		MesToggleWrite				: BOOL;					(* (NA) Cal: True := read authorised 	*)
		MesToggleRead				: BOOL;					(* (NA) Cal: True := Write authorised	*)
		                                    	                                                	
		
		
		
		
		
		
END_STRUCT
END_TYPE

// ---- 01_Equipement_Library/ProtectRelay/ProtectRelay_PACE100ST.TcDUT
TYPE ProtectRelay_PACE100ST :
STRUCT   
	
		Thermal_Overload			: REAL ; (* %  0 TO 250                         *)
	//Status                                 (*                                     *)
		Comut						: BOOL ; (* Cell's selector is in remote position    *)
		CB_Close					: BOOL ; (*  Cell is closes                                   *)
		CB_In_Alarm					: BOOL ; (*Cell is in alarm                                     *)
		Trip_Counter				: INT;   (*  Number of trip *)

                                  
		Mesdata 					: ProtectRelay;   (*                                     *)
        
END_STRUCT
END_TYPE

// ---- 01_Equipement_Library/ProtectRelay/ProtectRelay_REFIO.TcDUT
TYPE ProtectRelay_REFIO :
STRUCT
	
	MesData				: ProtectRelay ; 	(* Object 								    *)
	MesTransfoAlarm		: BOOL ; 	(* Transfo alarm                              *)
	MesSWOpened			: BOOL ;	(* Sectionneur de ligne ouvert              *)
	MesSWClosed			: BOOL ; 	(* Sectionneur de ligne fermé               *)
	MesEarth			: BOOL ; 	(* Earthing                                 *)
	MesSF6Low			: BOOL ; 	(* SF6 gaz is low                           *)
	MesSF6Unsufficient	: BOOL ; 	(* Sf6  is unsufficient                     *)
	MesTransfoWarning	: BOOL ; 	(* Transfo warning                            *)
	MesOpened			: BOOL ; 	(* Disjoncteur opened                       *)
	MesClosed			: BOOL ; 	(* Disjoncteur is closed                    *)
	MesComutLocal		: BOOL ; 	(* Commutateur Local/Distant.               *)
	
	
END_STRUCT
END_TYPE

// ---- 01_Equipement_Library/ProtectRelay/ProtectRelay_S42.TcDUT
TYPE ProtectRelay_S42 :
STRUCT
	
	MesData							: ProtectRelay ; 	(* Object *)

	MesAlarm_Phase1					: BOOL ;(* Default Phase 1*)		
	MesAlarm_Phase2				    : BOOL ;(*Default Phase 2*)
	MesAlarm_Phase3				    : BOOL ;(*Default Phase 3*)
	MesAlarm_PhaseRpt			    : BOOL ;(*Default Phase RPT (relai presence tension ? ) *)
	MesAlarm_Ground				    : BOOL ;(*Default Ground*)
	MesAlarm_GroundRpt			    : BOOL ;(*Default Ground RPT (relai presence tension ? )*)
	MesAlarm_MaxUInverse			: BOOL ;(*Default Max UI Inverse*)
	MesAlarm_MaxP				    : BOOL ;(*Default Max P *)
	MesAlarm_CB		   			 	: BOOL ;(*Default Circuit breaker *)
	MesAlarm_Watchdog				: BOOL ;(* Défault watchdog*)						
	OUT_CmdOpen	   			 		: BOOL ;(* Circuit breaker Open Command*)
	OUT_CmdClose	    			: BOOL ;(*Circuit breaker Close Command*) 
                      
	MesU0					    	: REAL ;(*(V) Residual Voltage*)
	MesP							: REAL ;(*(kW) Active Power*)
	MesQ							: REAL ;(*(kVAr) Reactive Power*)
	MesCosPhi						: REAL ;(*(p.u) CospPhi*)
	
	MesAlarm_CablesOvercharge 		: BOOL; (*Cables Overcharge*) 		
    MesAlarm_FaultFrom225kV			: BOOL; (*Fault From 225 kV*)		
	
	
END_STRUCT
END_TYPE

// ---- 01_Equipement_Library/ProtectRelay/ProtectRelay_S48.TcDUT
///////////
// Structure For I35. Main Operating Data to be saved ( ex: OPC ) .  
//////////
TYPE ProtectRelay_S48 :
STRUCT
	
		MesData						: ProtectRelay;			(*	(NA) Protection relay									    *)
                                                        	                                               
		                                    				                                                             
		MesU						: REAL;					(* (V) Average Phase to Phase Voltage                           *)
	                                                    	
		MesV1						: REAL ;        		(* (V) Average Phase to Phase Voltage                           *)
		MesV2						: REAL ;				(* (V) Average Phase to Phase Voltage                           *)
		MesV3						: REAL ;				(* (V) Average Phase to Phase Voltage                           *)
       			                                        	                   
		MesP						: REAL; 				(* (Kw)Power on Grid                                            *)
		MesQ						: REAL;					(* (kvar) Power on grid                                         *)
		MesS						: REAL;					(* (KVA) Power apparent                                         *)
		MesCosPhi					: REAL;					(* (NA) power factor                                            *)
		MesTanPhi					: REAL; 				(* (NA) Cal : tan Phi                                           *)
		   

                                 			                                                        
		MesStopPP_UminLong			: BOOL; 				(* (NA) PP is stopping during 2min, because of Long GTE fault	*)
		                                    			                                                          
		EActProd					: REAL; 				(* (MWh) Active Energy Produced                                 *)
		EActCons					: REAL; 				(* (MWh) Active Energy Consummed                                *)
		EReactProd					: REAL; 				(* (MVArh) Reactive Energy Produced                             *)
		EReactCons					: REAL; 				(* (MVArh) Reactive Energy Consummed                            *)
		                                    			                                                           
	// Relais Input                         			
		Input11						: BOOL;					(* (NA) Input 11 du relais de protection                        *)
		Input12                     : BOOL;					(* (NA) Input 12 du relais de protection                        *)
		Input13                     : BOOL;					(* (NA) Input 13 du relais de protection                        *)
		Input14                     : BOOL;					(* (NA) Input 14 du relais de protection                        *)
		Input21						: BOOL;					(* (NA) Input 21 du relais de protection                        *)
		Input22						: BOOL;					(* (NA) Input 22 du relais de protection                        *)
		Input23						: BOOL;					(* (NA) Input 23 du relais de protection                        *)
		Input24						: BOOL;					(* (NA) Input 24 du relais de protection                        *)
		Input25						: BOOL;					(* (NA) Input 25 du relais de protection                        *)
		Input26						: BOOL;					(* (NA) Input 26 du relais de protection                        *)
		
				
END_STRUCT
END_TYPE

// ---- 01_Equipement_Library/ProtectRelay/ProtectRelay_T20.TcDUT
///////////
// Structure For I35. Main Operating Data to be saved ( ex: OPC ) .  
//////////
TYPE ProtectRelay_T20 :
STRUCT
	// I35 Data measures
	
		MesData						: ProtectRelay; (*							*)							
                                           			(*                          *)
	                                       			(*                          *)
		MesFreq						: REAL;			(* (Hz) Frequence of grid   *)
		MesP						: REAL;			(* (Kw)Power on Grid        *)
		MesQ						: REAL;			(* (kvar) Power on grid     *)
		MesS						: REAL;			(* (KVA) Power apparent     *)
		                                   			(*                          *)
		MesTripProtec				: REAL;			(* A                        *)
		MesGlobalWarming		    : REAL;			(* % Au warming of TR       *)


END_STRUCT
END_TYPE

// ---- 01_Equipement_Library/ProtectRelay/ProtectRelay_T87.TcDUT
TYPE ProtectRelay_T87 :
STRUCT
	
	MesData							: ProtectRelay ; 		(* Object 								    *)

	MesAlarm_DiscordSectLigneHTB	: BOOL;   				(*DiscordSectLigneHTB*)
	MesAlarm_DiscordSectMaltHTB		: BOOL;   				(*DiscordSectMaltHTB	*)
	MesAlarm_DiscordSectDisjHTB		: BOOL;   				(*DiscordSectDisjHTB	*)
	MesAlarm_TeleCondamne			: BOOL;   				(*TeleCondamne		*)
	MesAlarm_DeTeleCondamne			: BOOL;   				(*DeTeleCondamne		*)
	MesAlarm_DiscordTeleCondamne	: BOOL;	  				(*DiscordTeleCondamne*)
                                                			
	MesAlarm_IoMaxCoteProd			: BOOL;   				(*IoMaxCoteProd*)
	MesAlarmUMax					: BOOL;   				(*UMax		*)
	MesAlarmUMax_Long				: BOOL;   				(*UMax_Long	*)
	MesAlarm_PhaseRpt				: BOOL;					(*PhaseRpt*)
	MesWarning_ImgTherm				: BOOL;					(*ImgTherm alarm*)
	MesAlarm_ImgTherm				: BOOL;					(*ImgTherm warning*)
	MesAlarm_DifferTransfo			: BOOL;					(*DifferTransfo*)
	MesAlarm_FreqMax				: BOOL;					(*FreqMax*)
	MesAlarm_FreqMin				: BOOL;					(*FreqMin*)	
	                                            			
	MesU0							: REAL;					(*(V) Residual Voltage*)
	MesP							: REAL;					(*(kW) Active Power*)	
	MesQ							: REAL;					(*(kVAr) Reactive Power*)
	

	
END_STRUCT
END_TYPE

// ---- 01_Equipement_Library/ProtectRelay/ProtectRelay_VIP410.TcDUT
TYPE ProtectRelay_VIP410 :
STRUCT
		MesData						: ProtectRelay; 	(* (NA) MesData 																												*)
		MesStatCom					: BOOL ; 			(* (NA) False: device did not respond successfully to most recent read or write request, True: device is responding normally	*)
		MesAvgI1					: REAL ; 			(* (A) Phase 1 Average current                                                                                       			*)
		MesAvgI2					: REAL ; 			(* (A) Phase 2 Average current                                                                                       			*)
		MesAvgI3					: REAL ; 			(* (A) Phase 3 Average current                                                                                       			*)
		MesI0Fault					: REAL ; 			(* (A) Fault current                                                                                                 			*)
		StatusWord					: WORD ; 			(* (NA) Status Word                                                                                                     		*)
		ControlWord					: WORD ; 			(* (NA) Control Word                                                                                                    		*)
END_STRUCT
END_TYPE

// ---- 01_Equipement_Library/ProtectRelay/ProtectRelay_WIP1.TcDUT
///////////
// Structure For I35. Main Operating Data to be saved ( ex: OPC ) .  
//////////
TYPE ProtectRelay_WIP1 :
STRUCT
	// I35 Data measures
	MesData					: ProtectRelay ; (**)


	
END_STRUCT
END_TYPE

// ---- 01_Equipement_Library/Router/Router.TcDUT
TYPE Router :
STRUCT
		MesWatchdog	        : BOOL ; 	(* Watchdog*)
		
		MesAlarmCode		: WORD ;	(* (NA) Internal Akuo AlarmCode		*)
		MesWarningCode		: WORD ; 	(* (NA) Internal Akuo WarningCode   *)
		MesEventCode		: WORD ; 	(* (NA) Internal Akuo EventCode	    *)
		
END_STRUCT
END_TYPE

// ---- 01_Equipement_Library/Router/Router_Standard.TcDUT
TYPE Router_Standard :
STRUCT
		MesData				: Router ;  (* Object *)

		
END_STRUCT
END_TYPE

// ---- 01_Equipement_Library/Sensors/ANA/ANA.TcDUT
TYPE ANA :
STRUCT
	Value 					: REAL ;	(* (-) Analogic Value 					*)
	                                    
	MesAlarmCode			: WORD ;	(* (NA) Internal Akuo AlarmCode     *)
	MesWarningCode			: WORD ;    (* (NA) Internal Akuo WarningCode   *)
	MesEventCode			: WORD ;    (* (NA) Internal Akuo EventCode		*)

END_STRUCT
END_TYPE

// ---- 01_Equipement_Library/Sensors/COM/AllInOne.TcDUT
TYPE AllInOne :
STRUCT
	
	MesWindSp 			: REAL ;		(* (m/s)	 Wind speed measurement of the weather station												        *)
	MesWindDir 			: REAL ;		(* (°) 		 Wind direction measurement of the weather station                                                  *)
	MesHygro			: REAL ;		(* (%) 		 Humidity measurement of the weather station                                                        *)
	MesTemp_Amb 			: REAL ;		(* (°C)		 Ambiant temperature measurement of the weather station                                             *)
	MesDewPoint			: REAL ;		(* (%) 		 Dew point measure of weather station                                                               *)
	MesRain1			: REAL ;		(* (count/h) Rain rate                                                                                          *)
	MesRain2			: REAL ;		(* (count/h) Rain rate                                                                                          *)
	MesRain3			: REAL ;		(* (count/h) Rain rate                                                                                          *)
                                        (*                                                                                                              *)
	MesAlarmWindSp		: REAL ;		(* Alarm for the Wind speed : 0=OFF, 1 = Lower threshold, 2 = Higher threshold                                  *)
	MesAlarmWindDir		: REAL ;		(* Alarm for the Wind direction : 0=OFF, 1 = Lower threshold, 2 = Higher threshold                              *)
	MesAlarmTemp		: REAL ;		(* Alarm for the temp sensor : 0=OFF, 1 = Lower threshold, 2 = Higher threshold                                 *)
	MesAlarmHygro		: REAL ;		(* Alarm for the humidity sensor : 0=OFF, 1 = Lower threshold, 2 = Higher threshold                             *)
	MesAlarmDewPt		: REAL ;		(* Alarm for the dew point sensor : 0=OFF, 1 = Lower threshold, 2 = Higher threshold                            *)
	MesAlarmRain1		: REAL ;		(* Alarm for the rain sensor : 0=OFF, 1 = Lower threshold, 2 = Higher threshold                                 *)
	MesAlarmRain2		: REAL ;		(* Alarm for the rain sensor : 0=OFF, 1 = Lower threshold, 2 = Higher threshold                                 *)
	MesAlarmRain3		: REAL ;		(* Alarm for the rain sensor : 0=OFF, 1 = Lower threshold, 2 = Higher threshold                                 *)
	                                    (*                                                                                                              *)
	MesAlarmCode		: WORD ;  	    (*                                                                                                              *)
	MesWarningCode		: WORD ;  	    (*                                                                                                              *)
	MesEventCode		: WORD ; 	    (*                                                                                                              *)
	
END_STRUCT
END_TYPE

// ---- 01_Equipement_Library/Sensors/COM/SMP1X.TcDUT
TYPE SMP1X :
STRUCT
	
	Value 						: REAL ;		(* (W/m²) Irradiance OF the pyranometer															*)
	Alarm						: REAL ;		(* Alarm for solar radiation (0=Off, 1 = Lower threshold, 2=Higher threshold)                   *)
	Description					: STRING ; 		(* Position and comments on the pyranometer                                                     *)
	                                            (*                                                                                              *)
	MesAlarmCode				: WORD ;  	    (*                                                                                              *)
	MesWarningCode				: WORD ;  	    (*                                                                                              *)
	MesEventCode				: WORD ; 	    (*                                                                                              *)
	
END_STRUCT
END_TYPE

// ---- 01_Equipement_Library/Sensors/TOR/TOR.TcDUT
TYPE TOR :
STRUCT
	
	MesAlarmState 		 		: BOOL  ;		(* TRUE = ALARM													*)
	MesCountAlarm				: UDINT ; 		(* Count the number of time the alarm has been triggered.       *)
                                                (*                                                              *)
	MesAlarmCode				: WORD ;		(* (NA) Internal Akuo AlarmCode                                 *)
	MesWarningCode				: WORD ;   	 	(* (NA) Internal Akuo WarningCode                               *)
	MesEventCode				: WORD ;	 	(* (NA) Internal Akuo EventCode		                            *)

END_STRUCT		
END_TYPE

// ---- 01_Equipement_Library/Sensors/TOR/TOR_Rain.TcDUT
TYPE TOR_Rain :
STRUCT
	
	MesData					: TOR ;		(* MesData 											 *)
	MesRainFall_LastHour  	: REAL;   	(* (mm)Amount of water fall during the last hour	 *)
	MesRainFall_LastDay   	: REAL;   	(* (mm)Amount of water fall during the last Day (mm) *)
	MesRainFall_LastMonth 	: REAL;   	(* (mm)Amour of water fall during the last Year (mm) *)
	                           
	AvgmmHour	  			: REAL; 	(* (mm)Hourly AVG of water fall                      *)
	AvgmmDay   				: REAL;     (* (mm)Daily AVG of water fall                       *)
	AvgmmMonth 				: REAL;     (* (mm) Monthly AVG of water fall                    *)
	
END_STRUCT
END_TYPE

// ---- 01_Equipement_Library/Sensors/TOR/TOR_Standard.TcDUT
TYPE TOR_Standard :
STRUCT
	
	MesData					: TOR ;		(* MesData 											 *)

END_STRUCT		
END_TYPE

// ---- 01_Equipement_Library/Tariff Meter/EM.TcDUT
TYPE EM :
STRUCT
	
	MesEActCons				: REAL ; 		(* Value of Active Energy consumed		*)
	MesEActProd				: REAL ;		(* Value of Active Energy produced      *)
	MesEReactCons			: REAL ;		(* Value of Reactive Energy consumed    *)
	MesEReactProd			: REAL ;		(* Value of Reactive Energy produced    *)
	                                                                             
	MesAlarmCode			: WORD ;	 	(* (NA) Internal Akuo AlarmCode         *)
	MesWarningCode			: WORD ; 		(* (NA) Internal Akuo WarningCode       *)
	MesEventCode			: WORD ; 		(* (NA) Internal Akuo EventCode	        *)

END_STRUCT
END_TYPE

// ---- 01_Equipement_Library/Tariff Meter/EM_Standard.TcDUT
TYPE EM_Standard :
STRUCT
	
	MesData			: EM ; 

END_STRUCT
END_TYPE

// ---- 01_Equipement_Library/Transfo/Transfo.TcDUT
TYPE Transfo :
STRUCT
    MesWarningTemp				: BOOL ;	(* Transfo Temperature warning		    *)
    MesAlarmTemp				: BOOL ;	(* Transfo Temperature Alarm		    *)
    MesAlarmGas					: BOOL ;	(* Transfo Gas Alarm			        *)
    MesAlarmOilLevel			: BOOL ;	(* Transfo Oil Level Alarm		        *)
    MesAlarmsSynthesis			: BOOL ;	(* Transfo Synthesis Alarm              *)
                                                                             
	MesAlarmCode				: WORD ;  	(* (NA) Internal Akuo AlarmCode         *)
	MesWarningCode				: WORD ; 	(* (NA) Internal Akuo WarningCode       *)
	MesEventCode				: WORD ; 	(* (NA) Internal Akuo EventCode	        *)

END_STRUCT
END_TYPE

// ---- 01_Equipement_Library/Transfo/Transfo_HV.TcDUT
TYPE Transfo_HV :
STRUCT

	MesData						: Transfo ; (* Transfo*)

	MesWarningGas					: BOOL  ; (* Buchholz warning*)

	MesWarning_TempLevel1			: BOOL  ; (*ImgTherm1erStade*)
	MesWarning_TempLevel2			: BOOL  ; (*ImgTherm2ndStade*)
	MesTrigger_Deletion				: BOOL  ; (*TransfoDcltSurpression*)

	MesTransfoRefrigLocal			: BOOL  ; (*TransfoRefrigLocal*)
	
	MesTrigger_NonReturnValve		: BOOL  ; (*declenchement clapet anti retour*)
	MesTrigger_ProtectRelay			: BOOL  ; (*DcltRelaisProtectRegl*)
	MesAlarm_TapChanger				: BOOL  ; (*Fault TapChanger*)
	
	


END_STRUCT
END_TYPE

// ---- 01_Equipement_Library/Transfo/Transfo_MV.TcDUT
TYPE Transfo_MV :
STRUCT
	
	MesData						: Transfo ; (* MesData *)


END_STRUCT
END_TYPE

// ---- 01_Equipement_Library/UPS/UPS.TcDUT
///////////
// Structure for UPS. Main Operating Data to be saved (ex: OPC)  
//////////
TYPE UPS :
STRUCT
		MesDischarging				: BOOL ; 			(* (NA) Battery is discharging		*)
		MesAlarm_Ulow				: BOOL ; 			(* (NA) Battery is almost empty     *)
		MesAlarmState				: BOOL ; 			(* (NA) Fault on the charger        *)
		MesUdc  					: REAL ; 			(* (V) DC Load voltage              *)
       		
		
		MesAlarmCode				: WORD ; 			(* Internal Akuo Alarm Code         *)
		MesWarningCode				: WORD ; 			(* Internal Akuo Warning Code       *)
		MesEventCode				: WORD ; 			(* Internal Akuo Warning Code 	    *)
        
		MesCP_Read					: BOOL := FALSE ;   (* Read function enable             *)
		MesAlarmCom					: BOOL ; 			(* Communication alarm              *)
	
END_STRUCT
END_TYPE

// ---- 01_Equipement_Library/UPS/UPS_CXC.TcDUT
///////////
// Structure For I35. Main Operating Data to be saved ( ex: OPC ) .  
//////////
TYPE UPS_CXC :
STRUCT
	
	MesData				: UPS ; 	(* Object 									*)
	            		            (*                                          *)
	MesU				: REAL ; 	(*(V) AC voltage                            *)
	MesIload			: REAL ; 	(*(A) DC Load current                       *)
	MesUBatt			: REAL ; 	(*(V) Battery voltage                       *)
	MesIBatt			: REAL ; 	(*(A) Battery Current                       *)
	MesSoC  			: REAL ; 	(*(%) Battery SoC                           *)
	MesIdc  			: REAL ; 	(*(A) battery + load Current                *)

	
	MesOverTempBatt 	: BOOL ; 	(* OverTemperature of the battery alarm		*)
	MesCBUpsOpened		: BOOL ; 	(* UPS CB opened alarm                      *)
	
		
	
END_STRUCT
END_TYPE

// ---- 01_Equipement_Library/UPS/UPS_ENERIS.TcDUT
///////////
// Structure For I35. Main Operating Data to be saved (ex: OPC).  
//////////
TYPE UPS_Eneris :
STRUCT
	// I35 Data measures
		MesData                     : UPS;  (* MesData *)
		
END_STRUCT
END_TYPE

// ---- 01_Equipement_Library/UPS/UPS_Eneris.TcDUT
///////////
// Structure For I35. Main Operating Data to be saved (ex: OPC).  
//////////
TYPE UPS_Eneris :
STRUCT
	// I35 Data measures
		MesData                     : UPS;  (* MesData *)
		
END_STRUCT
END_TYPE

// ---- 01_Equipement_Library/UPS/UPS_Eneris.TcDUT
///////////
// Structure For I35. Main Operating Data to be saved (ex: OPC).  
//////////
TYPE UPS_Eneris :
STRUCT
	// I35 Data measures
		MesData                     : UPS;  (* MesData *)
		
END_STRUCT
END_TYPE

// ---- 01_Equipement_Library/UPS/UPS_PS10048.TcDUT
///////////
// Structure for PS100_48. Main operating data to be saved (ex:OPC).  
//////////
TYPE UPS_PS10048 :
STRUCT
		MesData             : UPS; 			(* MesData 																		*)
		                            		                                                                                
		MesSoc				: REAL; 		(* (%) Battery charge indicator 												*)
		MesUdc_48V			: REAL; 		(* (V) 48V output voltage 														*)
		MesUdc_12V			: REAL; 		(* (V) 12V output voltage 														*)
		MesUBatt			: REAL; 		(* (V) 12V battery voltage	    												*)
		MesIdc_12V			: REAL; 		(* (A) 12V output current 														*)
		MesIdc_Bat			: REAL;			(* (A) Battery current 															*)
		                            		                                                                                
		MesDischarge		: REAL; 		(* (V) Serious discharge threshold 												*)
		MesEbackUp			: REAL; 		(* (%) Energy backup threshold 	   												*)
		MesCapacity_Nom		: REAL; 		(* (Ah) NomCapa 				   												*)
		                                                                       												
		MesEBackUpEna		: BOOL;  		(* (Na) Energy backup enabled 	   												*)
		MesBatTestPer		: BOOL;  		(* (Na) Battery test period 	  												*)
		MesVacTripSelect	: BOOL;  		(* (NA) 0: Low. Off = 52Vac, Low = 129Vac. 1: High. Off = 69Vac, Low = 172Vac	*)
		                                                                                                                    
		MesToggleWrite		: BOOL;			(* (NA) Cal : True = read authorised  											*)
		MesToggleRead		: BOOL;			(* (NA) Cal : True = Write authorised 											*)
		                           		                                                                                    
		MesAlarm_AcOff		: BOOL;			(* (NA) True = AC off 															*)
		MesAlarm_GeneralOff	: BOOL;			(* (NA) True = Imminent shutdown 												*)
	//	MesAlarm_LowBat		: BOOL;			(* (NA) True = discharge 														*)
		MesAlarm_AcLow		: BOOL;			(* (NA) True = AC power supply low 												*)
		                                                                                                                    
		MesFault_Minor		: BOOL;			(* (NA) True = Minor fault (overtemp, overcurrent, overvolt) 					*)
		MesFault_Major		: BOOL;			(* (NA) True = Major fault : cannot recover 									*)
		MesFault_Bat		: BOOL;			(* (NA) True = Battery disconnected 											*)
		MesFault_Charger	: BOOL;			(* (NA) True = Charger out of order 											*)
		MesFault_12V		: BOOL;			(* (NA) True = 12V absent 														*)
		MesFault_48V		: BOOL;			(* (NA) True = 48V absent 														*)
		                           	
END_STRUCT
END_TYPE

// ---- 04_Application/IO/IO.TcDUT
TYPE IO :
STRUCT
MesEventCode : ARRAY[1..7] OF WORD ; (*Akuo AlarmCode*)

END_STRUCT
END_TYPE

// ---- 04_Application/IO/ST_AI.TcDUT
TYPE ST_AI :
STRUCT
		Value		  AT %I*	: INT	;
		Description 			: STRING	;

END_STRUCT
END_TYPE

// ---- 04_Application/IO/ST_AO.TcDUT
TYPE ST_AO :
STRUCT
		Value		  AT %Q*	: INT	;
		Description 			: STRING	;

END_STRUCT
END_TYPE

// ---- 04_Application/IO/ST_DI.TcDUT
TYPE ST_DI :
STRUCT
		Value		  AT %I*	: BOOL	;
		Description 			: STRING	;

END_STRUCT
END_TYPE

// ---- 04_Application/IO/ST_DO.TcDUT
TYPE ST_DO :
STRUCT
		Value		  AT %Q*	: BOOL	;
		Description 			: STRING	;

END_STRUCT
END_TYPE

// ---- 00_FunctionsBlocks/Communication/IEC104/GVL_Cst.TcGVL
{attribute 'qualified_only'}
VAR_GLOBAL CONSTANT
		CstNbAOEntries			: INT :=  50 ;
END_VAR

// ---- 00_FunctionsBlocks/Fifo/GVL_Fifo.TcGVL
VAR_GLOBAL CONSTANT 
		Max_buffer_size_G					: UDINT:=10000000; // Max buffer size of fifo
END_VAR

// ---- 04_Application/CONFIG/GVL_BASE.TcGVL
///////////////////////
// DO NOT MODIFY :  
// Maximal number of objects  - Maximal array size 
////////////////////
VAR_GLOBAL CONSTANT 
	// PRODUCT 
	CstNbPTR_G					: BYTE := 4 ;  				// (NA) Number of PTR
	CstNbESS_G   				: BYTE := 3 ;  				// (NA) Number of ESS


	// EQUIPMENT
		//SUB_MV
	CstNbFeederMVCB_G			: BYTE	:= 3 ; 
		// PTR 
	CstNbInv_PTR_G				: BYTE := 2 ;				// Maximal Number of PV Inverters for PTR
	CstNbSB_INV_G				: BYTE := 32 ;				// Maximal Number of String box in inverter

		// EM 		
	CstNbEM_G					: BYTE := 1;				// Number of Energy Meters
		
		//ESS		
	CstNbPcs_ESS				: BYTE := 2  ;
	CstNbPowerCol_PCS_G			: BYTE := 3  ;				// Maximal Number of Power colonne by PCS
	CstNbHvac_ESS				: BYTE := 2  ;
	CstNbBank_Ess				: BYTE := 2  ;
	CstNbRack_BBMS				: BYTE := 2  ;
				
		
		//WS		
	CstNbPyrano					: UINT := 5;
	CstNbAnemo					: UINT := 1;
	CstNbPanTmp					: UINT := 4;
	CstNbAmbTmp					: UINT := 3;	
		
	// PP 
	CstNbCouplermax_G			: BYTE 	:= 100 ;			// Maximal number of ethercat devices 
	CstNbAlarmIO_G				: BYTE := 10 ; // Number of Event in PRG_IO.
	
	
	(*               SMS               							*)
	CstNbUser					: SINT:=10; //Nbr d'utilisateur utilisé par AX_Numtel
	CstNbCMD					: SINT:=20; //Nbr commande utilisé par AX_CMD_SMS
	CstNbAlarmCode				: INT:=213;  //Number of alarmcode use in AlarmManager
	
	// TIMEZONE
	    (* Indonesia East Standard Time Zone settings *)
        FRANCE_TZI : ST_TimeZoneInformation := (bias:=-60,
                                       		 				standardName:='Heure Française',
                                        					standardDate:=(wYear:=0,wMonth:=10,wDayOfWeek:=0,wDay:=27,wHour:=3),
                                        					standardBias:=0,
                                        					daylightName:='None',
                                        					daylightDate:=(wYear:=0,wMonth:=3,wDayOfWeek:=0,wDay:=31,wHour:=2),
                                        					daylightBias:=0);
			
		CstPhoneIndicator_G		: STRING := '+33';
			
		CstCycleTime_G			: INT := 10 ; 			// (ms) Cycle Time of the CPU . 

		CstNbRedundantVariableMax_G	: UINT := 553 ;
		CstNbParamOPCUA				: UINT := 100 ; 
	
END_VAR
VAR_GLOBAL
	sTimeGMT_G          	: STRING;				// Full Date Time for historization (GMT) 
	sTimeLocal_G		 	: STRING ;				// Local Time 
	CalGMTTimeStruct		: TIMESTRUCT ; 			// GMT Time Structure

	ParamOpenVpnFile		: STRING := '';			// Path to openvpn file. 
	ParamIpPublic 			: STRING(255);			// Public IP 
	MesSizeCdrive_PLC		: REAL := 100000 ; 		// (Mo) Remaining Disk space
	MesSizeCdrive_IndusPC	: REAL := 100000 ; 		// (Mo) Remaining Disk space
END_VAR

// ---- 04_Application/CONFIG/GVL_Beckhoff.TcGVL
VAR_GLOBAL
	CalLocalTimeStruct			: TIMESTRUCT;		// Local Time Structure
	CstTimeZone_G				: ST_TimeZoneInformation 	:= WEST_EUROPE_TZI ;	// Local TimeZone
	ParamDirBaseStore		: STRING := 'C:\TwinCAT\Functions\Historisation\';	// Directroy for the historization
	
	

	
END_VAR

// ---- 04_Application/CONFIG/GVL_CFG.TcGVL
///////////////
// Configuration Files. Define Power Plant sizing and references. 
//////////////
VAR_GLOBAL 
		CstPLCBackup 			: BOOL := FALSE ;  			// TRUE if this PLC is used as a backup . 
		CstNetAmsId_Slave		: STRING(20):= '5.49.202.22.1.1'; //NetAMSId Slave .'5.79.170.90.1.1'
		CstNetAmsId_IndusPC		: STRING(20):= ''; // set '' if no Indus PLC
		//CstIPIEC104			: STRING := '10.101.111.1' ; 
		
		
END_VAR
	
VAR_GLOBAL 
	// Solar Classique //
		A1_PP					: FB_PP  ;  								// MCA Power Plant 
 
	// PRODUCT DEFINITION //
		//PTR 
		AX_PTR 					: ARRAY[1..CstNbPTR_G] OF FB_PTR ; 	 		// Array with AMG products
		
		//SUB_MV
		A1_SUBMV				: FB_SUBMV ;	 					 		// SUB_MV		
		
		//WEATHER STATION
		A1_WS					: FB_WS;
		
		//ESS 
		//AX_ESS				: ARRAY[1..CstNbESS_G] OF FB_ESS ; 
		
	// GLOBAL VARIABLE //
	
		CmdClearFault_G			: BOOL ; 									// (NA) Clear all permanent faults
		CmdInit_G				: BOOL ; 									// (NA) Global Init Action
		CstIPIEC104				: STRING := '10.111.109.1' ; 		
END_VAR

// ---- 04_Application/CONFIG/GVL_Check.TcGVL
VAR_GLOBAL
	FaultCheck_G : BOOL ; // Test if Fault 
	Fault_Count_G: CTU  ; // Counter 	
	

END_VAR

// ---- 04_Application/CONFIG/GVL_DataBaseStructures.TcGVL
{attribute 'qualified_only'}
VAR_GLOBAL
	AX_StructModbusTCP 	AT %MW112 	: ARRAY[1..10000] OF WORD;
END_VAR

// ---- 04_Application/CONFIG/GVL_EmulConfig.TcGVL

VAR_GLOBAL CONSTANT 
	ParamVarAdsMax_G				: UINT := 82 ; // Maximum Object to exchange in Ads
END_VAR

VAR_GLOBAL
	
	ParamCycleTime_Emul				: REAL := 10 ; // Temps de reference d'emulation en ms . 

	MesFreqGen 						: REAL := 50;
	MesUGen							: REAL := 20600;
	ParamLossImpedance				: REAL := 0.000004 ; // Ohmic value to account for transfo losses . 2 10^-8 ohm.m * 200 m .
	
	MesP_INVmppt					: REAL := 2500; // MPPT Power for one inverter 
	
	SoCInit							: REAL := 50 ; 
 
	//////   IO ////// 
	MesTempExt: INT;
	MesWindDir: INT;
	MesWindSpd : INT ; 
	MesHygroExt: INT;
	MesPyra		: INT  ;
	// SuBMV 
	
	iCouplerStatePDL				: UINT ; 
	
	MeasureMVCB_Closed						: BOOL := TRUE; 
	MeasureMVCB_Opened						: BOOL ; 
	MeasureMVCB_Fuse						: BOOL ; 
	MeasureMVCB_Malt						: BOOL ; 
	

	MainMVCB_ComutLocal						: BOOL := TRUE; 
	MainMVCB_Malt						: BOOL ; 
	MainMVCB_Close						: BOOL;
	MainMVCB_Open						: BOOL ;
	
	FeederMVCBClose_External			: ARRAY[1..CstNbFeederMVCB_G] OF BOOL ; 
	FeederMVCBOpen_External			: ARRAY[1..CstNbFeederMVCB_G] OF BOOL ; 	

	FeederMVCB_ComutLocal		: ARRAY[1..CstNbFeederMVCB_G] OF BOOL ; 
	FeederMVCB_Malt		: ARRAY[1..CstNbFeederMVCB_G] OF BOOL ; 
	
	PDLEsState1_IO                : BOOL:=TRUE;
	PDLChainBESSState1_IO         : BOOL;
	PDLMainCBAuxState1_IO         : BOOL;
	PDLCB_SourceSwitch1State1_IO	:BOOL := TRUE; 
	PDLCB_SourceSwitch2State1_IO	:BOOL; 
	PDLCB_HTA1State1_IO           : BOOL;
	PDLCB_HTA2State1_IO           : BOOL;
	PDLCB_Rearmement1State1_IO    : BOOL;
	PDLCB_Rearmement2State1_IO    : BOOL;
	PDLIN_MesCbUPS_IO             : BOOL;    
	PDLFireSystemCBFSS_IO         : BOOL;
	PDLDsBTState1_IO              : BOOL;
	PDLDsHTState1_IO              : BOOL;
	PDLUPSFaultSynthesis_IO       : BOOL;  
	PDLUPSDischarging_IO          : BOOL;  
	PDLRPNWatchDog_IO             : BOOL := TRUE ;  
	PDLRPNWatchdogREU615_IO       : BOOL := TRUE  ;  
	PDLRPNAlarmIPos_IO            : BOOL;  
	PDLRPNAlarmVolt_IO				:BOOL; 
	
	PDLFireSystemWarning_IO			: BOOL;
	PDLFireSystemAlarm_IO			: BOOL;
	PDLFireSystemWatchdog_IO		: BOOL;
	
	
	
(*	
	// ESS
	MesTemp							: ARRAY[1..CstNbEss] OF ARRAY[1..4] OF INT;	
	MesHygr							: ARRAY[1..CstNbEss] OF ARRAY[1..4] OF INT;
	MesSpdState						: ARRAY[1..CstNbEss] OF BOOL;
	MesPcsDs						: ARRAY[1..CstNbEss] OF BOOL;
	MesBatDs						: ARRAY[1..CstNbEss] OF BOOL;
	MesToS							: ARRAY[1..CstNbEss] OF BOOL;
	Cb_Q31_Close					: ARRAY[1..CstNbEss] OF BOOL;
	Cb_Q31_Open						: ARRAY[1..CstNbEss] OF BOOL;
	MesPcs1Sd						: ARRAY[1..CstNbEss] OF BOOL;
	MesPcs2Sd						: ARRAY[1..CstNbEss] OF BOOL;
	MesEs							: ARRAY[1..CstNbEss] OF BOOL;
	Ds_Pcs							: ARRAY[1..CstNbEss] OF BOOL;
	Ds_Bat							: ARRAY[1..CstNbEss] OF BOOL;
	CmdReset_IO						: ARRAY[1..CstNbEss] OF BOOL;			
	MesUpsAlarm						: ARRAY[1..CstNbEss] OF BOOL;		
	MesUpsDischarging				: ARRAY[1..CstNbEss] OF BOOL;		
	MesSupplyFlt_40A_RC				: ARRAY[1..CstNbEss] OF BOOL;	
	MesSup_10A_PLC					: ARRAY[1..CstNbEss] OF BOOL;		
	bBatFireWarning					: ARRAY[1..CstNbEss] OF BOOL;
	bBatFireFault					: ARRAY[1..CstNbEss] OF BOOL;
	bBatFireAlarm					: ARRAY[1..CstNbEss] OF BOOL;
 	bDcSwitchBank1 					: ARRAY[1..CstNbEss] OF BOOL;
 	bDcSwitchBank2	 				: ARRAY[1..CstNbEss] OF BOOL;
 	bFanBank1	 					: ARRAY[1..CstNbEss] OF BOOL;
 	bFanBank2	 					: ARRAY[1..CstNbEss] OF BOOL;
	iCouplerState: ARRAY[1..CstNbESS]OF UINT;
	bCmdResetEss	 					: ARRAY[1..CstNbEss] OF BOOL;
	CoeffSuiviSetpointPcs			: REAL := 0.9;						// Pourcentage de suivi de la consigne à chaque pas de temps : si 1, MesPac = SetptP d'un pas de temps à l'autre, si 0 ne suit pas du tout le setpoint

*)
END_VAR

// ---- 04_Application/MAIN/MAIN_Emul.TcPOU
PROGRAM MAIN_Emul
VAR
	TP_1		: TP;
	TP_2		: TP;
	
	ClockReadIO				: BOOL;
	ClockReadCOM			: BOOL;
	//M_INIT VARIABLE //
		bInit					: BOOL := TRUE ;						// Initialization variable

		
		WriteAds		: ADSWRITE;
		bTest			: BOOL;
		
		
		// DATETIME //	
		FB_LocalSystTime      	: FB_LOCALSYSTEMTIME;	// Get time function
		FB_ToGMT : FB_TzSpecificLocalTimeToSystemTime;	// Local to UTC Time function
		TON_Time				: TON;
		CalLocalTimeStruct_Temp: TIMESTRUCT;
		//init
		FB_GetSystemTime        : GETSYSTEMTIME;						// GEt time function
		
		FB_ToLocal 				: FB_FileTimeToTzSpecificLocalTime;		// UTC to local Time function
		fileTime        		: T_FILETIME;							// Filetime format for UTC Time 
		FileTimeLocal			: T_FILETIME;							// Filetime format for local time		
		
		
		
		

END_VAR

VAR_OUTPUT
			OUT_CalRunningPLC_IO 		: BOOL ; 
END_VAR

	TP_1(IN:=NOT TP_1.Q , PT:= T#100MS);		// Pour les IO
	ClockReadIO 		:= TP_1.Q;
	TP_2(IN:=NOT TP_1.Q , PT:= T#1S);		// Pour la com
	ClockReadCOM 		:= TP_2.Q;

// INITIALIZATION//
	IF bInit OR CmdInit_G THEN

		M_Init() ; 
		bInit := FALSE; 
	END_IF
	

	TON_Time(IN:= TRUE, PT:=T#1200MS ) ; 
	FB_LocalSystTime(
		bEnable := TRUE,
		dwCycle := 1,
		systemTime => CalLocalTimeStruct_Temp);

	IF TON_Time.Q THEN 
		CalLocalTimeStruct:= CalLocalTimeStruct_Temp ; 
	END_IF
		
		FB_ToGMT(
		in	:= CalLocalTimeStruct,
		tzInfo := CstTimeZone_G,
		out	=> CalGMTTimeStruct);
	
	sTimeGMT_G	:= SYSTEMTIME_TO_STRING(CalGMTTimeStruct);
	sTimeLocal_G	:= SYSTEMTIME_TO_STRING(CalLocalTimeStruct);	

	
OUT_CalRunningPLC_IO := TRUE ; 

// INPUTS //

	PRG_IO() ; 	// Emul the IO
	PRG_IO.M_Inputs() ;  // On mets à jour les variables emulées pour l'ecriture

// PROGRAMMS CALLS //
		ADS_Custom();	// On execute le read et le write . 
	// Hybrid Power PLant 
		A1_PP();
	
	// Historization //
	PRG_IO.M_Outputs() ;  // On recupère les commandes IO. 
	
// OUTPUTS //

METHOD M_Init : BOOL
VAR_INPUT
END_VAR

VAR 
	Year : STRING ; 
	Month: STRING ; 
	Day : STRING ; 
	Hour: STRING ; 
	Str_Temp: STRING;
END_VAR
//CstCycleTime_G 		:= 50 ;							// Cycle Time
CstTimeZone_G 		:= WEST_EUROPE_TZI ; 		// Local Time Zone 
	



// Get the Windows time ( not accurate ) at startup before updating the system time. 
	// DateTime 
	
	
	FB_GetSystemTime(
		timeLoDW	=> fileTime.dwLowDateTime, 
		timeHiDW	=> fileTime.dwHighDateTime);
		
	FB_ToLocal(
		in			:=fileTime,
		tzInfo 		:= CstTimeZone_G,
		out		 	=> FileTimeLocal);
		
CalLocalTimeStruct := FILETIME_TO_SYSTEMTIME(FileTimelocal) ; 


Year := CONCAT(STR1:= WORD_TO_STRING(CalLocalTimeStruct.wYear), STR2:= '_') ; 
Month := CONCAT(STR1:= WORD_TO_STRING(CalLocalTimeStruct.wMonth), STR2:= '_') ;
Day := CONCAT(STR1:=WORD_TO_STRING(CalLocalTimeStruct.wDay), STR2:= ' ') ;
Hour := CONCAT(STR1:=WORD_TO_STRING(CalLocalTimeStruct.wHour), STR2:= 'h') ;

Str_Temp := Year ; 
Str_Temp := CONCAT(STR1:=Str_Temp , STR2:= Month )  ; 
Str_Temp := CONCAT(STR1:=Str_Temp , STR2:= Day )  ; 	
Str_Temp := CONCAT(STR1:=Str_Temp , STR2:= Hour )  ; 

A1_PP.MesData.MesStartTime 		:= Str_Temp  ; 	// Jour du dernier update de code .
END_METHOD

END_PROGRAM

// ---- 04_Application/IO/PRG_IO.TcPOU
PROGRAM PRG_IO
///////////
// This Program is used as an interface between code variable and the I/O cards
//////////
VAR_INPUT
	
//PP States //
	MesCouplerStateSUBMV		: ST_AI ; 

// EXECUTE VARIABLES //
	IN_CmdInhibOutput_OPC		: BOOL :=TRUE ; 
	
END_VAR
VAR 	
//M_INIT VARIABLES //
	bInit						: BOOL	:=TRUE ;			// Initialization variables
	iTest                       : INT;
END_VAR

VAR_INPUT
	KK : INT ;
	
	MesIO_SUBMV_EL1809_1 : ARRAY [1..16] OF ST_DI ; 
	MesIO_SUBMV_EL1809_2 : ARRAY [1..16] OF ST_DI ; 
	MesIO_SUBMV_EL1809_3 : ARRAY [1..16] OF ST_DI ;
	MesIO_SUBMV_EL1809_14 : ARRAY [1..16] OF ST_DI ; 
	MesIO_SUBMV_EL2809_4 : ARRAY [1..16] OF ST_DO ; 
	MesIO_SUBMV_EL3024_5 : ARRAY [1..4] OF ST_AI ; 
	MesIO_SUBMV_EL3024_12 : ARRAY [1..4]  OF ST_AI ;
	MesIO_SUBMV_EL3024_13 : ARRAY [1..4]  OF ST_AI ;
	MesIO_PTR_1_EL3024_8 : ARRAY [1..4] OF ST_AI ; 
	MesIO_PTR_1_EL1809_9 : ARRAY [1..16] OF ST_DI ; 
	MesIO_PTR_1_EL2809_10 : ARRAY [1..16] OF ST_DO ; 
	MesIO_PTR_2_EL3024_8 : ARRAY [1..4] OF ST_AI ; 
	MesIO_PTR_2_EL1809_9 : ARRAY [1..16] OF ST_DI ; 
	MesIO_PTR_2_EL2809_10 : ARRAY [1..16] OF ST_DO ; 
	MesIO_PTR_3_EL3024_8 : ARRAY [1..4] OF ST_AI ; 
	MesIO_PTR_3_EL1809_9 : ARRAY [1..16] OF ST_DI ; 
	MesIO_PTR_3_EL2809_10 : ARRAY [1..16] OF ST_DO ; 
	
END_VAR

// Initializing the static variables //  
	IF bInit OR CmdInit_G THEN
		M_Init() ; 
		bInit		:= FALSE ; 
	END_IF
	
	// EMULATOR OF IO 
	
	// On met ici les calculs pour émuler des variables IO qui ne serait pas liée à des commandes 

A1_SUBMV.IN_MesCouplerState_IO							:= iCouplerStatePDL ;
A1_SUBMV.A1_MeasureMVCB.IN_CmdExternalClose_Emul 		:=  MeasureMVCB_Closed ; 
A1_SUBMV.A1_MeasureMVCB.IN_CmdExternalOpen_Emul 		:=  MeasureMVCB_Opened ; 

FOR KK:= 1 TO CstNbFeederMVCB_G DO 
	A1_SUBMV.AX_FeederMVCB[KK].IN_CmdExternalClose_Emul := FeederMVCBClose_External[KK] ;
	A1_SUBMV.AX_FeederMVCB[KK].IN_CmdExternalOpen_Emul  := FeederMVCBOpen_External[KK] ;
	A1_SUBMV.AX_FeederMVCB[KK].IN_MesComutLocal_IO 		:=  FeederMVCB_ComutLocal[KK] ; 
	A1_SUBMV.AX_FeederMVCB[KK].IN_MesEarth_IO 			:=  FeederMVCB_Malt[KK]; 
END_FOR

// Close cells 
A1_SUBMV.A1_GridMVCB.IN_CmdExternalClose_Emul 		  := TRUE;
A1_SUBMV.A1_AuxMVCB.IN_CmdExternalClose_Emul   		  := TRUE;
A1_SUBMV.A1_MainMVCB.A1_Sect.IN_CmdExternalClose_Emul := TRUE; 


A1_SUBMV.A1_MeasureMVCB.IN_MesFuse_IO :=  MeasureMVCB_Fuse ; 
A1_SUBMV.A1_MeasureMVCB.IN_MesEarth_IO :=  MeasureMVCB_Malt ; 

IF A1_SUBMV.A1_MainMVCB.ParamComutNc THEN 
	A1_SUBMV.A1_MainMVCB.IN_MesComutLocal_IO :=  NOT MainMVCB_ComutLocal ; 
ELSE
	A1_SUBMV.A1_MainMVCB.IN_MesComutLocal_IO :=   MainMVCB_ComutLocal ;
END_IF

A1_SUBMV.A1_MainMVCB.IN_MesEarth_IO :=  MainMVCB_Malt ; 
A1_SUBMV.A1_MainMVCB.IN_CmdExternalClose_Emul	:= MainMVCB_Close ; 
A1_SUBMV.A1_MainMVCB.IN_CmdExternalOpen_Emul	:= MainMVCB_Open OR PDLRPNAlarmIPos_IO OR PDLRPNAlarmVolt_IO; 

A1_SUBMV.A1_ES_LV.IN_MesState1_IO                    := PDLEsState1_IO                   ;
A1_SUBMV.A1_ES_MV.IN_MesState1_IO                    := PDLEsState1_IO                   ;
A1_SUBMV.A1_MainCB_LV.IN_MesState1_IO                := PDLMainCBAuxState1_IO            ;

A1_SUBMV.A1_UPS_24v.IN_MesCbUPS_IO                   := PDLIN_MesCbUPS_IO                ;    
A1_SUBMV.A1_UPS_48v.IN_MesCbUPS_IO                   := PDLIN_MesCbUPS_IO                ;    

//A1_SUBMV.A1_SAFE_FireSystem.IN_MesCBFSS_IO            := PDLFireSystemCBFSS_IO         ;
A1_SUBMV.A1_DS_LV.IN_MesState1_IO                    := PDLDsBTState1_IO                 ;
A1_SUBMV.A1_DS_MV.IN_MesState1_IO                    := PDLDsHTState1_IO                 ;
A1_SUBMV.A1_UPS_24v.IN_MesFault_IO              	 := PDLUPSFaultSynthesis_IO          ; 
A1_SUBMV.A1_UPS_48v.IN_MesFault_IO              	 := PDLUPSFaultSynthesis_IO          ; 

A1_SUBMV.A1_ProtectRelay.IN_MesWatchDog_IO           := PDLRPNWatchDog_IO                ; 
A1_SUBMV.A1_ProtectRelay.IN_MesWatchDog_IO           := PDLRPNWatchdogREU615_IO          ; 
A1_SUBMV.A1_ProtectRelay.IN_MesAlarmIMax_IO          := PDLRPNAlarmIPos_IO               ; 
A1_SUBMV.A1_ProtectRelay.IN_MesAlarmUmin_IO			 := PDLRPNAlarmVolt_IO				;		

// WS 
A1_WS.A1_Temp_Ext.IN_MesValue1_IO	:= MesTempExt ; 
A1_WS.AX_Temp_Panel[1].IN_MesValue1_IO := MesTempExt;
A1_WS.A1_WindDir.IN_MesValue1_IO	:= MesWindDir ; 
A1_WS.A1_WindSp.IN_MesValue1_IO	:= MesWindSpd ; 

FOR KK:=1 TO CstNbPyrano DO 
	A1_WS.Ax_Pyrano[KK].IN_MesValue1_IO :=  MesPyra ; 
END_FOR 		




// ESS
(*	
FOR KK := 1 TO CstNbEss DO
	AX_ESS[KK].AX_TmpSensors[1].IN_MesValue_IO1 := MesTemp[KK][1];
	AX_ESS[KK].AX_HygroSensors[1].IN_MesValue_IO1 := MesHygr[KK][1];
	
	FOR LL := 2 TO 4 DO
		AX_ESS[KK].AX_TmpSensors[LL].IN_MesValue_IO1 := REAL_TO_INT(AX_ESS[KK].AX_HVAC[1].MesDataExd.MesData.MesTempRoom/50*32767) ; //MesTemp[KK][LL];
		AX_ESS[KK].AX_HygroSensors[LL].IN_MesValue_IO1 := REAL_TO_INT(AX_ESS[KK].AX_HVAC[1].MesDataExd.MesData.MesHygroAmb/100*32767) ;// MesHygr[KK][LL];
		
	END_FOR
	//MesIoESS_DI_1[KK][4].Value := GVL_EmulConfig.MesSpdState[KK];
	
	
	AX_Ess[KK].A1_Spd.IN_MesState1_IO 								:= 	MesSpdState[KK];						
	AX_ESS[KK].A1_Ds_Pcs.IN_MesState1_IO 							:=  MesPcsDs[KK];								
	AX_ESS[KK].A1_Ds_Bat.IN_MesState1_IO 							:=  MesBatDs[KK];								
	AX_ESS[KK].A1_ToS.IN_MesState1_IO 								:=  MesToS[KK];								
	AX_ESS[KK].A1_Cb_Q31.IN_CmdExternalClose_Emul							:=  Cb_Q31_Close[KK];							
	AX_ESS[KK].A1_Cb_Q31.IN_CmdExternalOpen_Emul 							:=  Cb_Q31_Open[KK];							
	AX_ESS[KK].A1_Sd_Pcs.IN_MesState1_IO 							:=  MesPcs1Sd[KK];							
	AX_ESS[KK].A1_Sd_Pcs.IN_MesState2_IO 							:=  MesPcs2Sd[KK];							
//	AX_ESS[KK].A1_Sd_Bat.IN_MesState1_IO 							:=  MesBat1Sd[KK];							
	AX_ESS[KK].A1_Es.IN_MesState1_IO 								:=  MesEs[KK];										
	AX_ESS[KK].A1_Ds_Pcs.IN_MesState1_IO 							:=  Ds_Pcs[KK];						
//	AX_ESS[KK].A1_Fuse1_Cab1.IN_MesState1_IO 						:=  Fuse1_Cab1[KK];						
//	AX_ESS[KK].A1_Fuse2_Cab1.IN_MesState1_IO 						:=  Fuse2_Cab1[KK];						
	AX_ESS[KK].A1_Ds_Bat.IN_MesState1_IO 							:=  Ds_Bat[KK];						
//	AX_ESS[KK].A1_Fuse1_Cab2.IN_MesState1_IO  						:=  Fuse1_Cab2[KK];						
//	AX_ESS[KK].A1_Fuse2_Cab2.IN_MesState1_IO  						:=  Fuse2_Cab2[KK];					
	AX_ESS[KK].IN_CmdReset_IO 										:=  CmdReset_IO[KK];				
	AX_ESS[KK].A1_UPS.IN_MesFaultSynthesis_IO						:=  MesUpsAlarm[KK];	
	AX_ESS[KK].A1_UPS.IN_MesDischarging_IO							:=  MesUpsDischarging[KK] ; 				
	AX_ESS[KK].A1_CB_PLC24V.IN_MesState1_IO					 		:=  MesSup_10A_PLC[KK];			
	AX_ESS[KK].A1_CB_RackCtrl24V.IN_MesState1_IO					:=  MesSupplyFlt_40A_RC[KK];			
	AX_ESS[KK].A1_FSS.IN_MesWarning_IO					 			:=  bBatFireWarning[KK];		
	AX_ESS[KK].A1_FSS.IN_MesFault_IO					 			:=  bBatFireFault[KK];	
	AX_ESS[KK].A1_FSS.IN_MesAlarm_IO					 			:=  bBatFireAlarm[KK];		
	AX_ESS[KK].AX_CB_ChainDcSwitchBank[1].IN_MesState1_IO           :=  bDcSwitchBank1[KK];		     
	AX_ESS[KK].AX_CB_ChainDcSwitchBank[2].IN_MesState1_IO           :=  bDcSwitchBank2[KK];	
	AX_ESS[KK].AX_CB_ChainFanBank[1].IN_MesState1_IO                :=  bFanBank1[KK];		     
	AX_ESS[KK].AX_CB_ChainFanBank[2].IN_MesState1_IO                :=  bFanBank2[KK];	   
	AX_ESS[KK].IN_MesCouplerState_IO								:= iCouplerState[KK] ;
	AX_ESS[KK].IN_CmdReset_IO										:= bCmdResetEss[KK] ; 	


END_FOR

	
*)

METHOD M_Init : BOOL
VAR
	KK : BYTE;
	
	LL: UINT ; 
	MM: INT;
	JJ: INT;
	
END_VAR

// WS
	MesTempExt	:= 16000 ; 
	MesWindDir     := 16000 ; 
	MesWindSpd     := 16000 ; 
	MesHygroExt	:= 16000 ; 
	MesPyra		:= 16000 ; 
// 
(*

FOR KK:= 1 TO CstNbESS_G DO 
	FOR LL:= 1 TO CstNbBank_Ess DO 
		FOR MM := 1 TO AX_ESS[KK].AX_Bbms[LL].ParamNbRacks DO
			FOR JJ := 1 TO AX_ESS[KK].AX_Bbms[LL].ParamNbRackString DO 
				MEMCPY(destAddr := ADR(AX_ESS[KK].AX_Bbms[LL].Rea.MesDataExd.MesData.AX_Rack[KK].AX_RACKSTRING[JJ].MesSoC) , srcAddr := ADR(SoCInit) , n:= SIZEOF(SoCInit)) ; 
			END_FOR
		END_FOR
	END_FOR
END_FOR


iCouplerStatePDL :=  8 ; 

PDLChainBESSState1_IO := TRUE ;
FOR KK := 1 TO CstNbEss DO
	FOR LL := 1 TO 4 DO
			 MesTemp[KK][LL] := 16000 ;		//32767 ma value 
			MesHygr[KK][LL] := 16000;
		
	END_FOR
	//MesIoESS_DI_1[KK][4].Value := GVL_EmulConfig.MesSpdState[KK];
	
	
MesSpdState[KK]					:= FALSE ;			
MesPcsDs[KK]					:= FALSE ;				
MesBatDs[KK]					:= FALSE ;				
MesToS[KK]						:= TRUE ;			
Cb_Q31_Close[KK]				:= TRUE ;				
Cb_Q31_Open[KK]					:= FALSE ;				
MesPcs1Sd[KK]					:= FALSE ;			
MesPcs2Sd[KK]					:= FALSE ;			
MesEs[KK]						:= FALSE ;					
Ds_Pcs[KK]						:= FALSE ;	
Ds_Bat[KK]						:= FALSE ;	
CmdReset_IO[KK]					:= FALSE ;	
MesUpsAlarm[KK]	        		:= FALSE ;
MesUpsDischarging[KK] 			:= FALSE ;			
MesSup_10A_PLC[KK]				:= TRUE ;
MesSupplyFlt_40A_RC[KK]			:= TRUE ;		
bBatFireWarning[KK]				:= FALSE ;
bBatFireFault[KK]        		:= FALSE ;
bBatFireAlarm[KK]	    		:= FALSE ;
bDcSwitchBank1[KK]	    		:= FALSE ; 
bDcSwitchBank2[KK]      	 	:= FALSE ;
bFanBank1[KK]		        	:= TRUE ;
bFanBank2[KK]   				:= TRUE ;
iCouplerState[KK]				:= 8 ;
END_FOR
		*)
END_METHOD

METHOD M_Inputs
///////////
// Intput interface between POUs and I/O Cards
//////////////

VAR 
KK							: BYTE ; 					// For LOOP 
MesCouplerStateSUB_MV			: ST_AI ; 
END_VAR

MesIO_SUBMV_EL1809_1[ 1].value  			:= A1_SUBMV.AX_FeederMVCB[1].IN_MesOpened_IO 	;	
MesIO_SUBMV_EL1809_1[ 2].value        		:=   A1_SUBMV.AX_FeederMVCB[2].IN_MesOpened_IO	;
MesIO_SUBMV_EL1809_1[ 3].value        	:=   A1_SUBMV.AX_FeederMVCB[3].IN_MesOpened_IO	;	
MesIO_SUBMV_EL1809_1[ 4].value        		:=   A1_SUBMV.A1_MainMVCB.IN_MesOpened_IO		;
MesIO_SUBMV_EL1809_1[ 5].value        		:=   A1_SUBMV.A1_MainMVCB.IN_MesTripped_IO		;
MesIO_SUBMV_EL1809_1[ 6].value        		:=   A1_SUBMV.A1_MainMVCB.IN_MesEarth_IO  		;
MesIO_SUBMV_EL1809_1[ 7].value        		:=   A1_SUBMV.A1_MainMVCB.IN_MesComutLocal_IO	;
MesIO_SUBMV_EL1809_1[ 8].value        		:=   A1_SUBMV.A1_MainMVCB.IN_MesAlarmPwr_IO		;
MesIO_SUBMV_EL1809_1[ 9].value        		:=   A1_SUBMV.AX_FeederMVCB[1].IN_MesTripped_IO	;
MesIO_SUBMV_EL1809_1[ 10].value    			:=   A1_SUBMV.AX_FeederMVCB[2].IN_MesTripped_IO	;	
MesIO_SUBMV_EL1809_1[ 11].value    		:=   A1_SUBMV.AX_FeederMVCB[3].IN_MesTripped_IO	;  
MesIO_SUBMV_EL1809_1[ 12].value    			:=   A1_SUBMV.AX_FeederMVCB[1].IN_MesAlarmPwr_IO;  	
MesIO_SUBMV_EL1809_1[ 13].value    			:=   A1_SUBMV.AX_FeederMVCB[2].IN_MesAlarmPwr_IO;  	
MesIO_SUBMV_EL1809_1[ 14].value    		:=   A1_SUBMV.AX_FeederMVCB[3].IN_MesAlarmPwr_IO;  
MesIO_SUBMV_EL1809_1[ 15].value    			:=   A1_SUBMV.AX_FeederMVCB[1].IN_MesEarth_IO	;  
MesIO_SUBMV_EL1809_1[ 16].value    			:=   A1_SUBMV.AX_FeederMVCB[2].IN_MesEarth_IO	;  
MesIO_SUBMV_EL1809_2[ 1].value     		:=   A1_SUBMV.AX_FeederMVCB[3].IN_MesEarth_IO	;  
MesIO_SUBMV_EL1809_2[ 2].value     			:=   A1_SUBMV.AX_FeederMVCB[1].IN_MesComutLocal_IO;   
MesIO_SUBMV_EL1809_2[ 3].value     			:=   A1_SUBMV.AX_FeederMVCB[2].IN_MesComutLocal_IO;   
MesIO_SUBMV_EL1809_2[ 4].value    		:= A1_SUBMV.AX_FeederMVCB[3].IN_MesComutLocal_IO ;
MesIO_SUBMV_EL1809_2[ 5].value       		:=   A1_SUBMV.A1_GridMVCB.IN_MesOpened_IO			 ;		
MesIO_SUBMV_EL1809_2[ 6].value       		:=   A1_SUBMV.A1_MeasureMVCB.IN_MesOpened_IO		 ;		
MesIO_SUBMV_EL1809_2[ 7].value       		:=   A1_SUBMV.A1_MeasureMVCB.IN_MesFuse_IO  		 ;		
MesIO_SUBMV_EL1809_2[ 8].value       		:=   A1_SUBMV.A1_MeasureMVCB.IN_MesEarth_IO 		 ;		
MesIO_SUBMV_EL1809_2[ 9].value       		:=   A1_SUBMV.A1_AuxMVCB.IN_MesOpened_IO			 ; 			
MesIO_SUBMV_EL1809_2[ 10].value       		:=   A1_SUBMV.A1_AuxMVCB.IN_MesFuse_IO				 ;
MesIO_SUBMV_EL1809_2[ 11].value       		:=   A1_SUBMV.A1_AuxMVCB.IN_MesEarth_IO				 ;
MesIO_SUBMV_EL1809_2[ 12].value       		:=   A1_SUBMV.A1_ES_LV.IN_MesState1_IO				 ;
MesIO_SUBMV_EL1809_2[ 13].value       		:=   A1_SUBMV.A1_ES_MV.IN_MesState1_IO				 ;
MesIO_SUBMV_EL1809_2[ 14].value       		:=   A1_SUBMV.A1_SD_LV.IN_MesState1_IO				 ;
MesIO_SUBMV_EL1809_2[ 15].value       		:=   A1_SUBMV.A1_SD_MV.IN_MesState1_IO				 ;
MesIO_SUBMV_EL1809_2[ 16].value       		:=   A1_SUBMV.A1_Transfo_Aux.IN_MesAlarmsSynthesis_IO;
MesIO_SUBMV_EL1809_3[ 1].value 				:= 	 A1_SUBMV.A1_MainMVCB.A1_Sect.IN_MesClosed_IO 	 ;    
MesIO_SUBMV_EL1809_3[ 2].value       		:=   A1_SUBMV.A1_Transfo_Aux.IN_MesAlarmGas_IO		 ; 
MesIO_SUBMV_EL1809_3[ 3].value       		:=   A1_SUBMV.A1_Transfo_Aux.IN_MesWarningTemp_IO	 ; 
MesIO_SUBMV_EL1809_3[ 4].value       		:=   A1_SUBMV.A1_Transfo_Aux.IN_MesAlarmTemp_IO		 ; 
MesIO_SUBMV_EL1809_3[ 5].value       		:=   A1_SUBMV.A1_UPS_24v.IN_MesDischarging_IO		 ; 
MesIO_SUBMV_EL1809_3[ 6].value       		:=   A1_SUBMV.A1_UPS_24v.IN_MesFault_IO				 ; 
MesIO_SUBMV_EL1809_3[ 7].value       		:=   A1_SUBMV.A1_UPS_24v.IN_MesBatLow_IO			 ; 
MesIO_SUBMV_EL1809_3[ 8].value       		:=   A1_SUBMV.A1_ProtectRelay.IN_MesAlarmIMax_IO	 ; 
MesIO_SUBMV_EL1809_14[ 6].value       		:=   A1_SUBMV.A1_ProtectRelay.IN_MesAlarmUmin_IO	 ; 
MesIO_SUBMV_EL3024_5[ 1].value       		:=   A1_WS.Ax_Pyrano[1].IN_MesValue1_IO				 ; 
MesIO_SUBMV_EL3024_5[ 2].value       		:=   A1_WS.Ax_Pyrano[2].IN_MesValue1_IO				 ; 
MesIO_SUBMV_EL3024_5[ 3].value       		:=   A1_WS.A1_Temp_Ext.IN_MesValue1_IO				 ; 
MesIO_SUBMV_EL3024_5[ 4].value       		:=   A1_WS.A1_Hygro_Ext.IN_MesValue1_IO				 ; 
MesIO_SUBMV_EL3024_13[ 1].value       		:=   A1_WS.A1_WindDir.IN_MesValue1_IO				 ; 
MesIO_SUBMV_EL3024_13[ 2].value       		:=   A1_WS.A1_WindSp.IN_MesValue1_IO				 ; 
MesIO_PTR_1_EL3024_8[ 1].value       		:=   A1_WS.AX_Temp_Panel[1].IN_MesValue1_IO			 ; 
MesIO_PTR_1_EL3024_8[ 2].value       		:=   A1_WS.AX_Temp_Panel[1].IN_MesValue2_IO			 ; 
MesIO_PTR_1_EL3024_8[ 3].value       		:=   A1_WS.Ax_Pyrano[3].IN_MesValue1_IO				 ; 
MesIO_PTR_1_EL1809_9[ 1].value       		:=   AX_PTR[1].A1_MainMVCB_PTR.IN_MesAlarmPwr_IO 	 ; 
MesIO_PTR_1_EL1809_9[ 2].value       		:=   AX_PTR[1].A1_MainMVCB_PTR.IN_MesTripped_IO		 ; 
MesIO_PTR_1_EL1809_9[ 3].value       		:=   AX_PTR[1].A1_MainMVCB_PTR.IN_MesComutLocal_IO	 ; 
MesIO_PTR_1_EL1809_9[ 4].value       		:=   AX_PTR[1].A1_MainMVCB_PTR.IN_MesEarth_IO		 ; 
MesIO_PTR_1_EL1809_9[ 5].value       		:=   AX_PTR[1].A1_SD_Transfo.IN_MesState1_IO		 ; 
MesIO_PTR_1_EL1809_9[ 6].value       		:=   AX_PTR[1].A1_SD_INV.IN_MesState1_IO			 ; 
MesIO_PTR_1_EL1809_9[ 7].value       		:=   AX_PTR[1].A1_DS_Transfo.IN_MesState1_IO		 ; 
MesIO_PTR_1_EL1809_9[ 8].value       		:=   AX_PTR[1].A1_DS_INV.IN_MesState1_IO			 ; 
MesIO_PTR_1_EL1809_9[ 9].value       		:=   AX_PTR[1].A1_Transfo.IN_MesAlarmsSynthesis_IO	 ; 
MesIO_PTR_1_EL1809_9[ 11].value      		:=   AX_PTR[1].A1_Transfo.IN_MesAlarmGas_IO			 ;
MesIO_PTR_1_EL1809_9[ 12].value      		:=   AX_PTR[1].A1_Transfo.IN_MesWarningTemp_IO		 ;
MesIO_PTR_1_EL1809_9[ 13].value      		:=   AX_PTR[1].A1_Transfo.IN_MesAlarmTemp_IO		 ;
MesIO_PTR_1_EL1809_9[ 14].value      		:=   AX_PTR[1].A1_MainCBAux.IN_MesState1_IO			 ;
MesIO_PTR_2_EL3024_8[ 1].value       		:=   A1_WS.AX_Temp_Panel[2].IN_MesValue1_IO			 ; 
MesIO_PTR_2_EL3024_8[ 2].value       		:=   A1_WS.AX_Temp_Panel[2].IN_MesValue2_IO			 ; 
MesIO_PTR_2_EL3024_8[ 3].value       		:=   A1_WS.Ax_Pyrano[4].IN_MesValue1_IO				 ; 
MesIO_PTR_2_EL1809_9[ 1].value       		:=   AX_PTR[2].A1_MainMVCB_PTR.IN_MesAlarmPwr_IO	 ;  
MesIO_PTR_2_EL1809_9[ 2].value       		:=   AX_PTR[2].A1_MainMVCB_PTR.IN_MesTripped_IO 	 ; 
MesIO_PTR_2_EL1809_9[ 3].value       		:=   AX_PTR[2].A1_MainMVCB_PTR.IN_MesComutLocal_IO	 ; 
MesIO_PTR_2_EL1809_9[ 4].value       		:=   AX_PTR[2].A1_MainMVCB_PTR.IN_MesEarth_IO		 ; 
MesIO_PTR_2_EL1809_9[ 5].value       		:=   AX_PTR[2].A1_SD_Transfo.IN_MesState1_IO 		 ; 
MesIO_PTR_2_EL1809_9[ 6].value       		:=   AX_PTR[2].A1_SD_INV.IN_MesState1_IO			 ; 
MesIO_PTR_2_EL1809_9[ 7].value       		:=   AX_PTR[2].A1_DS_Transfo.IN_MesState1_IO		 ; 
MesIO_PTR_2_EL1809_9[ 8].value       		:=   AX_PTR[2].A1_DS_INV.IN_MesState1_IO			 ; 
MesIO_PTR_2_EL1809_9[ 9].value       		:=   AX_PTR[2].A1_Transfo.IN_MesAlarmsSynthesis_IO	 ; 
MesIO_PTR_2_EL1809_9[ 11].value      		:=   AX_PTR[2].A1_Transfo.IN_MesAlarmGas_IO			 ; 
MesIO_PTR_2_EL1809_9[ 12].value      		:=   AX_PTR[2].A1_Transfo.IN_MesWarningTemp_IO		 ; 
MesIO_PTR_2_EL1809_9[ 13].value      		:=   AX_PTR[2].A1_Transfo.IN_MesAlarmTemp_IO		 ; 
MesIO_PTR_2_EL1809_9[ 14].value      		:=   AX_PTR[2].A1_MainCBAux.IN_MesState1_IO 		 ; 
MesIO_PTR_3_EL3024_8[ 1].value       		:=   A1_WS.AX_Temp_Panel[3].IN_MesValue1_IO 		 ; 
MesIO_PTR_3_EL3024_8[ 2].value       		:=   A1_WS.AX_Temp_Panel[3].IN_MesValue2_IO 		 ; 
MesIO_PTR_3_EL3024_8[ 3].value       		:=   A1_WS.Ax_Pyrano[5].IN_MesValue1_IO				 ; 
MesIO_PTR_3_EL1809_9[ 1].value       		:=   AX_PTR[3].A1_MainMVCB_PTR.IN_MesAlarmPwr_IO	 ; 
MesIO_PTR_3_EL1809_9[ 2].value       		:=   AX_PTR[3].A1_MainMVCB_PTR.IN_MesTripped_IO		 ; 
MesIO_PTR_3_EL1809_9[ 3].value       		:=   AX_PTR[3].A1_MainMVCB_PTR.IN_MesComutLocal_IO	 ; 
MesIO_PTR_3_EL1809_9[ 4].value       		:=   AX_PTR[3].A1_MainMVCB_PTR.IN_MesEarth_IO		 ; 
MesIO_PTR_3_EL1809_9[ 5].value       		:=   AX_PTR[3].A1_SD_Transfo.IN_MesState1_IO		 ; 
MesIO_PTR_3_EL1809_9[ 6].value       		:=   AX_PTR[3].A1_SD_INV.IN_MesState1_IO			 ; 
MesIO_PTR_3_EL1809_9[ 7].value       		:=   AX_PTR[3].A1_DS_Transfo.IN_MesState1_IO		 ; 
MesIO_PTR_3_EL1809_9[ 8].value       		:=   AX_PTR[3].A1_DS_INV.IN_MesState1_IO			 ; 
MesIO_PTR_3_EL1809_9[ 9].value       		:=   AX_PTR[3].A1_Transfo.IN_MesAlarmsSynthesis_IO	 ; 
MesIO_PTR_3_EL1809_9[ 11].value       		:=   AX_PTR[3].A1_Transfo.IN_MesAlarmGas_IO			 ;
MesIO_PTR_3_EL1809_9[ 12].value       		:=   AX_PTR[3].A1_Transfo.IN_MesWarningTemp_IO		 ;
MesIO_PTR_3_EL1809_9[ 13].value       		:=   AX_PTR[3].A1_Transfo.IN_MesAlarmTemp_IO		 ;
MesIO_PTR_3_EL1809_9[ 14].value       		:=   AX_PTR[3].A1_MainCBAux.IN_MesState1_IO			 ;

MesIO_SUBMV_EL1809_3[ 9].value				:= 	A1_SUBMV.A1_GRID.IN_CmdAutCpl_IO			 	  	; 
MesIO_SUBMV_EL1809_3[ 10].value 			:= 	A1_SUBMV.A1_GRID.IN_CmdDisconnect_End_IO		  	; 
MesIO_SUBMV_EL1809_3[ 11].value 			:= 	A1_SUBMV.A1_GRID.IN_CmdDisconnect_IO			  	; 
MesIO_SUBMV_EL1809_3[ 12].value 			:= 	A1_SUBMV.A1_GRID.IN_CmdRSEOn_IO					  	; 
MesIO_SUBMV_EL1809_3[ 13].value 			:= 	A1_SUBMV.A1_GRID.IN_CmdRSEOff_IO				  	; 
MesIO_SUBMV_EL1809_3[ 14].value 			:= 	A1_SUBMV.A1_GRID.IN_CmdTAOn_IO 					  	; 
MesIO_SUBMV_EL1809_3[ 15].value 			:= 	A1_SUBMV.A1_GRID.IN_CmdTAOff_IO					  	; 
MesIO_SUBMV_EL1809_3[ 16].value 			:= 	A1_SUBMV.A1_GRID.IN_CmdStopPReg_IO 				  	; 

MesIO_SUBMV_EL1809_14[ 1].value 			:= 	A1_SUBMV.A1_GRID.IN_CmdStartPReg_IO				  	; 
MesIO_SUBMV_EL1809_14[ 2].value 			:= 	A1_SUBMV.A1_GRID.IN_CmdStopQReg_IO 				  	; 
MesIO_SUBMV_EL1809_14[ 3].value 			:= 	A1_SUBMV.A1_GRID.IN_CmdStartQReg_IO				  	; 
MesIO_SUBMV_EL1809_14[ 4].value 			:= 	A1_SUBMV.A1_GRID.IN_CmdEmergencyDisconnect_End_IO	; 
MesIO_SUBMV_EL1809_14[ 5].value 			:= 	A1_SUBMV.A1_GRID.IN_CmdEmergencyDisconnect_IO	  	; 

MesIO_SUBMV_EL3024_12[ 1].value             :=  A1_SUBMV.A1_GRID.IN_MesP0Reg_IO; 
MesIO_SUBMV_EL3024_12[ 2].value 			:=  A1_SUBMV.A1_GRID.IN_MesQ0Reg_IO;
END_METHOD

METHOD M_Outputs : BOOL
///////////
// Intput interface between POUs and I/O Cards
//////////////
VAR
	KK	: BYTE;

END_VAR

MEMCPY( destAddr  :=  ADR(A1_SUBMV.A1_MainMVCB.OUT_CmdOpen_IO  )		, SrcAddr :=  ADR(MesIO_SUBMV_EL2809_4[ 1].value ), n:= SIZEOF(MesIO_SUBMV_EL2809_4[ 1].value ) ) ; 				
MEMCPY( destAddr  :=  ADR(A1_SUBMV.A1_MainMVCB.OUT_CmdClose_IO )		, SrcAddr :=  ADR(MesIO_SUBMV_EL2809_4[ 2].value ), n:= SIZEOF(MesIO_SUBMV_EL2809_4[ 2].value ) ) ; 				
MEMCPY( destAddr  :=  ADR(A1_SUBMV.AX_FeederMVCB[1].OUT_CmdClose_IO )	, SrcAddr :=  ADR(MesIO_SUBMV_EL2809_4[ 3].value ), n:= SIZEOF(MesIO_SUBMV_EL2809_4[ 3].value ) ) ; 				
MEMCPY( destAddr  :=  ADR(A1_SUBMV.AX_FeederMVCB[2].OUT_CmdClose_IO )	, SrcAddr :=  ADR(MesIO_SUBMV_EL2809_4[ 4].value ), n:= SIZEOF(MesIO_SUBMV_EL2809_4[ 4].value ) ) ; 				
//MEMCPY( destAddr  :=  ADR(A1_SUBMV.AX_FeederMVCB[3].OUT_CmdClose_IO )	, SrcAddr :=  ADR(MesIO_SUBMV_EL2809_4[ 5].value ), n:= SIZEOF(MesIO_SUBMV_EL2809_4[ 5].value ) ) ; 				
MEMCPY( destAddr  :=  ADR(A1_SUBMV.AX_FeederMVCB[1].OUT_CmdOpen_IO )	, SrcAddr :=  ADR(MesIO_SUBMV_EL2809_4[ 6].value ), n:= SIZEOF(MesIO_SUBMV_EL2809_4[ 6].value ) ) ; 				
MEMCPY( destAddr  :=  ADR(A1_SUBMV.AX_FeederMVCB[2].OUT_CmdOpen_IO )	, SrcAddr :=  ADR(MesIO_SUBMV_EL2809_4[ 7].value ), n:= SIZEOF(MesIO_SUBMV_EL2809_4[ 7].value ) ) ; 				
//MEMCPY( destAddr  :=  ADR(A1_SUBMV.AX_FeederMVCB[3].OUT_CmdOpen_IO )	, SrcAddr :=  ADR(MesIO_SUBMV_EL2809_4[ 8].value ), n:= SIZEOF(MesIO_SUBMV_EL2809_4[ 8].value ) ) ; 				
MEMCPY( destAddr  :=  ADR(AX_PTR[1].A1_MainMVCB_PTR.OUT_CmdOpen_IO )	, SrcAddr :=  ADR(MesIO_PTR_1_EL2809_10[ 1].value), n:= SIZEOF(MesIO_PTR_1_EL2809_10[ 1].value) ) ; 				
MEMCPY( destAddr  :=  ADR(AX_PTR[1].A1_MainMVCB_PTR.OUT_CmdClose_IO )	, SrcAddr :=  ADR(MesIO_PTR_1_EL2809_10[ 2].value), n:= SIZEOF(MesIO_PTR_1_EL2809_10[ 2].value) ) ; 				
MEMCPY( destAddr  :=  ADR(AX_PTR[2].A1_MainMVCB_PTR.OUT_CmdOpen_IO )	, SrcAddr :=  ADR(MesIO_PTR_2_EL2809_10[ 1].value), n:= SIZEOF(MesIO_PTR_2_EL2809_10[ 1].value) ) ; 				
MEMCPY( destAddr  :=  ADR(AX_PTR[2].A1_MainMVCB_PTR.OUT_CmdClose_IO )	, SrcAddr :=  ADR(MesIO_PTR_2_EL2809_10[ 2].value), n:= SIZEOF(MesIO_PTR_2_EL2809_10[ 2].value) ) ; 				
MEMCPY( destAddr  :=  ADR(AX_PTR[3].A1_MainMVCB_PTR.OUT_CmdOpen_IO )	, SrcAddr :=  ADR(MesIO_PTR_3_EL2809_10[ 1].value), n:= SIZEOF(MesIO_PTR_3_EL2809_10[ 1].value) ) ; 				
MEMCPY( destAddr  :=  ADR(AX_PTR[3].A1_MainMVCB_PTR.OUT_CmdClose_IO )	, SrcAddr :=  ADR(MesIO_PTR_3_EL2809_10[ 2].value), n:= SIZEOF(MesIO_PTR_3_EL2809_10[ 2].value) ) ; 				


// Use NOT instead of X_end variable for Grid Disconnect/EmergencyDisconnect, example: 
//MesIO_SUBMV_EL2624_8[ 1].value 	:= NOT A1_SUBMV.A1_GRID.OUT_MesEmergencyDisconnect_IO AND NOT IN_CmdInhibOutput_OPC;
END_METHOD

END_PROGRAM

// ---- 04_Application/ADS/ADS_Custom.TcPOU
PROGRAM ADS_Custom

VAR_INPUT PERSISTENT
	ParamVarAds				: UINT := 82 ; // Number of ADS variable to exchange 
	ParamPortPrincipal 		: UINT := 851 ; // ADS Port of the main code  
END_VAR

VAR
	
bAlarmADSSize				: BOOL;		// Raise an alarm if one structure has a different size on the emulator than on the main code. 


ReadAds						: ARRAY[1..ParamVarAdsMax_G ] OF  Adsread ;
WriteAds					: ARRAY[1..ParamVarAdsMax_G ] OF  AdsWrite ;
KK							: UINT ; 
PLC_ReadSymInfoByName 		: ARRAY[1..ParamVarAdsMax_G] OF PLC_ReadSymInfoByName ;
SignalName 					: ARRAY[1..ParamVarAdsMax_G] OF STRING ; 	// Tableau des noms de variable à aller chercher sur le code principal
Address						: ARRAY[1..ParamVarAdsMax_G] OF PVOID ;	// Tableau des adresses mémoires de la variable sur l'émulator
bClockIO					: ARRAY[1..ParamVarAdsMax_G] OF BOOL ; // If True , update every 100 ms , else every 1 sec . 

Taille						: ARRAY[1..ParamVarAdsMax_G] OF PVOID ;	// Tableau de la taille pris par la variable sur l'émulatOR  
ReadAdsType					: ARRAY[1..ParamVarAdsMax_G] OF BOOL ; 	// Tableau pour savoir si la variable doit etre importé vers l'emulator
WriteAdsType				: ARRAY[1..ParamVarAdsMax_G] OF BOOL ; //  Tableau pour savoir si la variable doit etre exporté vers le code principal
CP_Read						: ARRAY[1..ParamVarAdsMax_G] OF BOOL ; 	// Condition de lecture ou d'ecriture ads


BInit						: BOOL:= TRUE;

END_VAR

IF BInit THEN 
	M_Init();
END_IF

bAlarmADSSize := FALSE; 
FOR KK:= 1 TO MIN(ParamVarAds, ParamVarAdsMax_G) DO 
	// Get Infos only if output is empty
	IF PLC_ReadSymInfoByName[KK].SYMINFO.symEntryLen = 0 OR bInit THEN
		PLC_ReadSymInfoByName[KK](NETid := '', Port:=ParamPortPrincipal,Symname:=SignalName[KK], Start:= CalLocalTimeStruct.wSecond= KK MOD 60 OR bInit,TMOUT:= T#5S) ;
	END_IF
	
	CP_Read[KK] := SEL( bClockIO[KK] ,MAIN_Emul.ClockReadCOM , MAIN_Emul.ClockReadIO)  AND NOT (PLC_ReadSymInfoByName[KK].SYMINFO.idxOffset=0) AND NOT PLC_ReadSymInfoByName[KK].ERR AND NOT ReadAds[KK].BUSY  ; 

	// Control that Source and destination Structure have the same size. 
	IF  PLC_ReadSymInfoByName[KK].SYMINFO.byteSize <> Taille[KK] THEN 
		bAlarmADSSize := TRUE; 
	END_IF

	// Read signal 
	IF ReadAdsType[KK] AND (PLC_ReadSymInfoByName[KK].SYMINFO.byteSize = Taille[KK]) THEN 
	
		ReadAds[KK](NETID:='',
					   PORT:=ParamPortPrincipal,
					   IDXGRP:=	PLC_ReadSymInfoByName[KK].SYMINFO.idxGroup,
					   IDXOFFS:=PLC_ReadSymInfoByName[KK].SYMINFO.idxOffset,
					   LEN:=PLC_ReadSymInfoByName[KK].SYMINFO.byteSize,
					   READ:=CP_Read[KK],
					   DESTADDR:=Address[KK], 
					   TMOUT:= T#100MS);
					   
	ELSIF WriteAdsType[KK] AND (PLC_ReadSymInfoByName[KK].SYMINFO.byteSize = Taille[KK]) THEN 
		WriteAds[KK]
		(
			NETID := '',
			PORT := ParamPortPrincipal,
			IDXGRP := PLC_ReadSymInfoByName[KK].SYMINFO.idxGroup,
			IDXOFFS := PLC_ReadSymInfoByName[KK].SYMINFO.idxOffset,
			LEN := PLC_ReadSymInfoByName[KK].SYMINFO.byteSize,
			SRCADDR := Address[KK],
			WRITE := CP_Read[KK],
			TMOUT := T#100MS
		);					   
	END_IF		   	   
END_FOR

bInit:= FALSE ;

METHOD M_Init
VAR_INPUT
END_VAR
SignalName[1]:='GVL_CFG.AX_PTR[1].A1_Datalogger.MesDataExd';	bClockIO[1]:=FALSE;	Taille[1]:=SIZEOF(GVL_CFG.AX_PTR[1].A1_Datalogger.MesDataExd);	Address[1]:=ADR(GVL_CFG.AX_PTR[1].A1_Datalogger.MesDataExd);	ReadAdsType[1]:=FALSE;	WriteAdsType[1]:=TRUE;
SignalName[2]:='GVL_CFG.AX_PTR[2].A1_Datalogger.MesDataExd';	bClockIO[2]:=FALSE;	Taille[2]:=SIZEOF(GVL_CFG.AX_PTR[2].A1_Datalogger.MesDataExd);	Address[2]:=ADR(GVL_CFG.AX_PTR[2].A1_Datalogger.MesDataExd);	ReadAdsType[2]:=FALSE;	WriteAdsType[2]:=TRUE;
SignalName[3]:='GVL_CFG.AX_PTR[3].A1_Datalogger.MesDataExd';	bClockIO[3]:=FALSE;	Taille[3]:=SIZEOF(GVL_CFG.AX_PTR[3].A1_Datalogger.MesDataExd);	Address[3]:=ADR(GVL_CFG.AX_PTR[3].A1_Datalogger.MesDataExd);	ReadAdsType[3]:=FALSE;	WriteAdsType[3]:=TRUE;
SignalName[4]:='GVL_CFG.AX_PTR[4].A1_Datalogger.MesDataExd';	bClockIO[4]:=FALSE;	Taille[4]:=SIZEOF(GVL_CFG.AX_PTR[4].A1_Datalogger.MesDataExd);	Address[4]:=ADR(GVL_CFG.AX_PTR[4].A1_Datalogger.MesDataExd);	ReadAdsType[4]:=FALSE;	WriteAdsType[4]:=TRUE;
SignalName[5]:='GVL_CFG.AX_PTR[1].A1_Datalogger.CmdbyCom';	bClockIO[5]:=FALSE;	Taille[5]:=SIZEOF(GVL_CFG.AX_PTR[1].A1_Datalogger.CmdbyCom);	Address[5]:=ADR(GVL_CFG.AX_PTR[1].A1_Datalogger.CmdbyCom);	ReadAdsType[5]:=TRUE;	WriteAdsType[5]:=FALSE;
SignalName[6]:='GVL_CFG.AX_PTR[2].A1_Datalogger.CmdbyCom';	bClockIO[6]:=FALSE;	Taille[6]:=SIZEOF(GVL_CFG.AX_PTR[2].A1_Datalogger.CmdbyCom);	Address[6]:=ADR(GVL_CFG.AX_PTR[2].A1_Datalogger.CmdbyCom);	ReadAdsType[6]:=TRUE;	WriteAdsType[6]:=FALSE;
SignalName[7]:='GVL_CFG.AX_PTR[3].A1_Datalogger.CmdbyCom';	bClockIO[7]:=FALSE;	Taille[7]:=SIZEOF(GVL_CFG.AX_PTR[3].A1_Datalogger.CmdbyCom);	Address[7]:=ADR(GVL_CFG.AX_PTR[3].A1_Datalogger.CmdbyCom);	ReadAdsType[7]:=TRUE;	WriteAdsType[7]:=FALSE;
SignalName[8]:='GVL_CFG.AX_PTR[4].A1_Datalogger.CmdbyCom';	bClockIO[8]:=FALSE;	Taille[8]:=SIZEOF(GVL_CFG.AX_PTR[4].A1_Datalogger.CmdbyCom);	Address[8]:=ADR(GVL_CFG.AX_PTR[4].A1_Datalogger.CmdbyCom);	ReadAdsType[8]:=TRUE;	WriteAdsType[8]:=FALSE;
SignalName[9]:='GVL_CFG.AX_PTR[1].AX_INV[1].MesDataExd';	bClockIO[9]:=FALSE;	Taille[9]:=SIZEOF(GVL_CFG.AX_PTR[1].AX_INV[1].MesDataExd);	Address[9]:=ADR(GVL_CFG.AX_PTR[1].AX_INV[1].MesDataExd);	ReadAdsType[9]:=FALSE;	WriteAdsType[9]:=TRUE;
SignalName[10]:='GVL_CFG.AX_PTR[1].AX_INV[2].MesDataExd';	bClockIO[10]:=FALSE;	Taille[10]:=SIZEOF(GVL_CFG.AX_PTR[1].AX_INV[2].MesDataExd);	Address[10]:=ADR(GVL_CFG.AX_PTR[1].AX_INV[2].MesDataExd);	ReadAdsType[10]:=FALSE;	WriteAdsType[10]:=TRUE;
SignalName[11]:='GVL_CFG.AX_PTR[2].AX_INV[1].MesDataExd';	bClockIO[11]:=FALSE;	Taille[11]:=SIZEOF(GVL_CFG.AX_PTR[2].AX_INV[1].MesDataExd);	Address[11]:=ADR(GVL_CFG.AX_PTR[2].AX_INV[1].MesDataExd);	ReadAdsType[11]:=FALSE;	WriteAdsType[11]:=TRUE;
SignalName[12]:='GVL_CFG.AX_PTR[2].AX_INV[2].MesDataExd';	bClockIO[12]:=FALSE;	Taille[12]:=SIZEOF(GVL_CFG.AX_PTR[2].AX_INV[2].MesDataExd);	Address[12]:=ADR(GVL_CFG.AX_PTR[2].AX_INV[2].MesDataExd);	ReadAdsType[12]:=FALSE;	WriteAdsType[12]:=TRUE;
SignalName[13]:='GVL_CFG.AX_PTR[3].AX_INV[1].MesDataExd';	bClockIO[13]:=FALSE;	Taille[13]:=SIZEOF(GVL_CFG.AX_PTR[3].AX_INV[1].MesDataExd);	Address[13]:=ADR(GVL_CFG.AX_PTR[3].AX_INV[1].MesDataExd);	ReadAdsType[13]:=FALSE;	WriteAdsType[13]:=TRUE;
SignalName[14]:='GVL_CFG.AX_PTR[3].AX_INV[2].MesDataExd';	bClockIO[14]:=FALSE;	Taille[14]:=SIZEOF(GVL_CFG.AX_PTR[3].AX_INV[2].MesDataExd);	Address[14]:=ADR(GVL_CFG.AX_PTR[3].AX_INV[2].MesDataExd);	ReadAdsType[14]:=FALSE;	WriteAdsType[14]:=TRUE;
SignalName[15]:='GVL_CFG.AX_PTR[4].AX_INV[1].MesDataExd';	bClockIO[15]:=FALSE;	Taille[15]:=SIZEOF(GVL_CFG.AX_PTR[4].AX_INV[1].MesDataExd);	Address[15]:=ADR(GVL_CFG.AX_PTR[4].AX_INV[1].MesDataExd);	ReadAdsType[15]:=FALSE;	WriteAdsType[15]:=TRUE;
SignalName[16]:='GVL_CFG.AX_PTR[4].AX_INV[2].MesDataExd';	bClockIO[16]:=FALSE;	Taille[16]:=SIZEOF(GVL_CFG.AX_PTR[4].AX_INV[2].MesDataExd);	Address[16]:=ADR(GVL_CFG.AX_PTR[4].AX_INV[2].MesDataExd);	ReadAdsType[16]:=FALSE;	WriteAdsType[16]:=TRUE;
SignalName[17]:='GVL_CFG.AX_PTR[1].AX_INV[1].ClockRead';	bClockIO[17]:=TRUE;	Taille[17]:=SIZEOF(GVL_CFG.AX_PTR[1].AX_INV[1].ClockRead);	Address[17]:=ADR(GVL_CFG.AX_PTR[1].AX_INV[1].ClockRead);	ReadAdsType[17]:=TRUE;	WriteAdsType[17]:=FALSE;
SignalName[18]:='GVL_CFG.AX_PTR[1].AX_INV[2].ClockRead';	bClockIO[18]:=TRUE;	Taille[18]:=SIZEOF(GVL_CFG.AX_PTR[1].AX_INV[2].ClockRead);	Address[18]:=ADR(GVL_CFG.AX_PTR[1].AX_INV[2].ClockRead);	ReadAdsType[18]:=TRUE;	WriteAdsType[18]:=FALSE;
SignalName[19]:='GVL_CFG.AX_PTR[2].AX_INV[1].ClockRead';	bClockIO[19]:=TRUE;	Taille[19]:=SIZEOF(GVL_CFG.AX_PTR[2].AX_INV[1].ClockRead);	Address[19]:=ADR(GVL_CFG.AX_PTR[2].AX_INV[1].ClockRead);	ReadAdsType[19]:=TRUE;	WriteAdsType[19]:=FALSE;
SignalName[20]:='GVL_CFG.AX_PTR[2].AX_INV[2].ClockRead';	bClockIO[20]:=TRUE;	Taille[20]:=SIZEOF(GVL_CFG.AX_PTR[2].AX_INV[2].ClockRead);	Address[20]:=ADR(GVL_CFG.AX_PTR[2].AX_INV[2].ClockRead);	ReadAdsType[20]:=TRUE;	WriteAdsType[20]:=FALSE;
SignalName[21]:='GVL_CFG.AX_PTR[3].AX_INV[1].ClockRead';	bClockIO[21]:=TRUE;	Taille[21]:=SIZEOF(GVL_CFG.AX_PTR[3].AX_INV[1].ClockRead);	Address[21]:=ADR(GVL_CFG.AX_PTR[3].AX_INV[1].ClockRead);	ReadAdsType[21]:=TRUE;	WriteAdsType[21]:=FALSE;
SignalName[22]:='GVL_CFG.AX_PTR[3].AX_INV[2].ClockRead';	bClockIO[22]:=TRUE;	Taille[22]:=SIZEOF(GVL_CFG.AX_PTR[3].AX_INV[2].ClockRead);	Address[22]:=ADR(GVL_CFG.AX_PTR[3].AX_INV[2].ClockRead);	ReadAdsType[22]:=TRUE;	WriteAdsType[22]:=FALSE;
SignalName[23]:='GVL_CFG.AX_PTR[4].AX_INV[1].ClockRead';	bClockIO[23]:=TRUE;	Taille[23]:=SIZEOF(GVL_CFG.AX_PTR[4].AX_INV[1].ClockRead);	Address[23]:=ADR(GVL_CFG.AX_PTR[4].AX_INV[1].ClockRead);	ReadAdsType[23]:=TRUE;	WriteAdsType[23]:=FALSE;
SignalName[24]:='GVL_CFG.AX_PTR[4].AX_INV[2].ClockRead';	bClockIO[24]:=TRUE;	Taille[24]:=SIZEOF(GVL_CFG.AX_PTR[4].AX_INV[2].ClockRead);	Address[24]:=ADR(GVL_CFG.AX_PTR[4].AX_INV[2].ClockRead);	ReadAdsType[24]:=TRUE;	WriteAdsType[24]:=FALSE;
SignalName[25]:='GVL_CFG.AX_PTR[1].AX_INV[1].ClockWrite';	bClockIO[25]:=TRUE;	Taille[25]:=SIZEOF(GVL_CFG.AX_PTR[1].AX_INV[1].ClockWrite);	Address[25]:=ADR(GVL_CFG.AX_PTR[1].AX_INV[1].ClockWrite);	ReadAdsType[25]:=TRUE;	WriteAdsType[25]:=FALSE;
SignalName[26]:='GVL_CFG.AX_PTR[1].AX_INV[2].ClockWrite';	bClockIO[26]:=TRUE;	Taille[26]:=SIZEOF(GVL_CFG.AX_PTR[1].AX_INV[2].ClockWrite);	Address[26]:=ADR(GVL_CFG.AX_PTR[1].AX_INV[2].ClockWrite);	ReadAdsType[26]:=TRUE;	WriteAdsType[26]:=FALSE;
SignalName[27]:='GVL_CFG.AX_PTR[2].AX_INV[1].ClockWrite';	bClockIO[27]:=TRUE;	Taille[27]:=SIZEOF(GVL_CFG.AX_PTR[2].AX_INV[1].ClockWrite);	Address[27]:=ADR(GVL_CFG.AX_PTR[2].AX_INV[1].ClockWrite);	ReadAdsType[27]:=TRUE;	WriteAdsType[27]:=FALSE;
SignalName[28]:='GVL_CFG.AX_PTR[2].AX_INV[2].ClockWrite';	bClockIO[28]:=TRUE;	Taille[28]:=SIZEOF(GVL_CFG.AX_PTR[2].AX_INV[2].ClockWrite);	Address[28]:=ADR(GVL_CFG.AX_PTR[2].AX_INV[2].ClockWrite);	ReadAdsType[28]:=TRUE;	WriteAdsType[28]:=FALSE;
SignalName[29]:='GVL_CFG.AX_PTR[3].AX_INV[1].ClockWrite';	bClockIO[29]:=TRUE;	Taille[29]:=SIZEOF(GVL_CFG.AX_PTR[3].AX_INV[1].ClockWrite);	Address[29]:=ADR(GVL_CFG.AX_PTR[3].AX_INV[1].ClockWrite);	ReadAdsType[29]:=TRUE;	WriteAdsType[29]:=FALSE;
SignalName[30]:='GVL_CFG.AX_PTR[3].AX_INV[2].ClockWrite';	bClockIO[30]:=TRUE;	Taille[30]:=SIZEOF(GVL_CFG.AX_PTR[3].AX_INV[2].ClockWrite);	Address[30]:=ADR(GVL_CFG.AX_PTR[3].AX_INV[2].ClockWrite);	ReadAdsType[30]:=TRUE;	WriteAdsType[30]:=FALSE;
SignalName[31]:='GVL_CFG.AX_PTR[4].AX_INV[1].ClockWrite';	bClockIO[31]:=TRUE;	Taille[31]:=SIZEOF(GVL_CFG.AX_PTR[4].AX_INV[1].ClockWrite);	Address[31]:=ADR(GVL_CFG.AX_PTR[4].AX_INV[1].ClockWrite);	ReadAdsType[31]:=TRUE;	WriteAdsType[31]:=FALSE;
SignalName[32]:='GVL_CFG.AX_PTR[4].AX_INV[2].ClockWrite';	bClockIO[32]:=TRUE;	Taille[32]:=SIZEOF(GVL_CFG.AX_PTR[4].AX_INV[2].ClockWrite);	Address[32]:=ADR(GVL_CFG.AX_PTR[4].AX_INV[2].ClockWrite);	ReadAdsType[32]:=TRUE;	WriteAdsType[32]:=FALSE;
SignalName[33]:='GVL_CFG.A1_SUBMV.A1_ProtectRelay.MesDataExd';	bClockIO[33]:=FALSE;	Taille[33]:=SIZEOF(GVL_CFG.A1_SUBMV.A1_ProtectRelay.MesDataExd);	Address[33]:=ADR(GVL_CFG.A1_SUBMV.A1_ProtectRelay.MesDataExd);	ReadAdsType[33]:=FALSE;	WriteAdsType[33]:=TRUE;
SignalName[34]:='GVL_CFG.A1_SUBMV.A1_ProtectRelay.ClockRead';	bClockIO[34]:=TRUE;	Taille[34]:=SIZEOF(GVL_CFG.A1_SUBMV.A1_ProtectRelay.ClockRead);	Address[34]:=ADR(GVL_CFG.A1_SUBMV.A1_ProtectRelay.ClockRead);	ReadAdsType[34]:=TRUE;	WriteAdsType[34]:=FALSE;
SignalName[35]:='GVL_CFG.A1_SUBMV.A1_PM.MesDataExd';	bClockIO[35]:=FALSE;	Taille[35]:=SIZEOF(GVL_CFG.A1_SUBMV.A1_PM.MesDataExd);	Address[35]:=ADR(GVL_CFG.A1_SUBMV.A1_PM.MesDataExd);	ReadAdsType[35]:=FALSE;	WriteAdsType[35]:=TRUE;
SignalName[36]:='GVL_CFG.A1_SUBMV.A1_PM.ClockRead';	bClockIO[36]:=TRUE;	Taille[36]:=SIZEOF(GVL_CFG.A1_SUBMV.A1_PM.ClockRead);	Address[36]:=ADR(GVL_CFG.A1_SUBMV.A1_PM.ClockRead);	ReadAdsType[36]:=TRUE;	WriteAdsType[36]:=FALSE;
SignalName[37]:='GVL_CFG.A1_SUBMV.A1_PM_Aux.MesDataExd';	bClockIO[37]:=FALSE;	Taille[37]:=SIZEOF(GVL_CFG.A1_SUBMV.A1_PM_Aux.MesDataExd);	Address[37]:=ADR(GVL_CFG.A1_SUBMV.A1_PM_Aux.MesDataExd);	ReadAdsType[37]:=FALSE;	WriteAdsType[37]:=TRUE;
SignalName[38]:='GVL_CFG.A1_SUBMV.A1_PM_Aux.ClockRead';	bClockIO[38]:=TRUE;	Taille[38]:=SIZEOF(GVL_CFG.A1_SUBMV.A1_PM_Aux.ClockRead);	Address[38]:=ADR(GVL_CFG.A1_SUBMV.A1_PM_Aux.ClockRead);	ReadAdsType[38]:=TRUE;	WriteAdsType[38]:=FALSE;
SignalName[39]:='GVL_CFG.A1_SUBMV.A1_UPS_48v.ClockRead';	bClockIO[39]:=TRUE;	Taille[39]:=SIZEOF(GVL_CFG.A1_SUBMV.A1_UPS_48v.ClockRead);	Address[39]:=ADR(GVL_CFG.A1_SUBMV.A1_UPS_48v.ClockRead);	ReadAdsType[39]:=TRUE;	WriteAdsType[39]:=FALSE;
SignalName[40]:='GVL_CFG.A1_SUBMV.A1_UPS_24v.ClockRead';	bClockIO[40]:=TRUE;	Taille[40]:=SIZEOF(GVL_CFG.A1_SUBMV.A1_UPS_24v.ClockRead);	Address[40]:=ADR(GVL_CFG.A1_SUBMV.A1_UPS_24v.ClockRead);	ReadAdsType[40]:=TRUE;	WriteAdsType[40]:=FALSE;
SignalName[41]:='PRG_IO.MesCouplerStateSUBMV';	bClockIO[41]:=TRUE;	Taille[41]:=SIZEOF(PRG_IO.MesCouplerStateSUBMV);	Address[41]:=ADR(PRG_IO.MesCouplerStateSUBMV);	ReadAdsType[41]:=FALSE;	WriteAdsType[41]:=TRUE;
SignalName[42]:='PRG_IO.MesIO_SUBMV_EL1809_1';	bClockIO[42]:=TRUE;	Taille[42]:=SIZEOF(PRG_IO.MesIO_SUBMV_EL1809_1);	Address[42]:=ADR(PRG_IO.MesIO_SUBMV_EL1809_1);	ReadAdsType[42]:=FALSE;	WriteAdsType[42]:=TRUE;
SignalName[43]:='PRG_IO.MesIO_SUBMV_EL1809_2';	bClockIO[43]:=TRUE;	Taille[43]:=SIZEOF(PRG_IO.MesIO_SUBMV_EL1809_2);	Address[43]:=ADR(PRG_IO.MesIO_SUBMV_EL1809_2);	ReadAdsType[43]:=FALSE;	WriteAdsType[43]:=TRUE;
SignalName[44]:='PRG_IO.MesIO_SUBMV_EL1809_3';	bClockIO[44]:=TRUE;	Taille[44]:=SIZEOF(PRG_IO.MesIO_SUBMV_EL1809_3);	Address[44]:=ADR(PRG_IO.MesIO_SUBMV_EL1809_3);	ReadAdsType[44]:=FALSE;	WriteAdsType[44]:=TRUE;
SignalName[45]:='PRG_IO.MesIO_SUBMV_EL2809_4';	bClockIO[45]:=TRUE;	Taille[45]:=SIZEOF(PRG_IO.MesIO_SUBMV_EL2809_4);	Address[45]:=ADR(PRG_IO.MesIO_SUBMV_EL2809_4);	ReadAdsType[45]:=TRUE;	WriteAdsType[45]:=FALSE;
SignalName[46]:='PRG_IO.MesIO_SUBMV_EL3024_5';	bClockIO[46]:=TRUE;	Taille[46]:=SIZEOF(PRG_IO.MesIO_SUBMV_EL3024_5);	Address[46]:=ADR(PRG_IO.MesIO_SUBMV_EL3024_5);	ReadAdsType[46]:=FALSE;	WriteAdsType[46]:=TRUE;
SignalName[47]:='PRG_IO.MesIO_PTR_1_EL3024_8';	bClockIO[47]:=TRUE;	Taille[47]:=SIZEOF(PRG_IO.MesIO_PTR_1_EL3024_8);	Address[47]:=ADR(PRG_IO.MesIO_PTR_1_EL3024_8);	ReadAdsType[47]:=FALSE;	WriteAdsType[47]:=TRUE;
SignalName[48]:='PRG_IO.MesIO_PTR_1_EL1809_9';	bClockIO[48]:=TRUE;	Taille[48]:=SIZEOF(PRG_IO.MesIO_PTR_1_EL1809_9);	Address[48]:=ADR(PRG_IO.MesIO_PTR_1_EL1809_9);	ReadAdsType[48]:=FALSE;	WriteAdsType[48]:=TRUE;
SignalName[49]:='PRG_IO.MesIO_PTR_1_EL2809_10';	bClockIO[49]:=TRUE;	Taille[49]:=SIZEOF(PRG_IO.MesIO_PTR_1_EL2809_10);	Address[49]:=ADR(PRG_IO.MesIO_PTR_1_EL2809_10);	ReadAdsType[49]:=TRUE;	WriteAdsType[49]:=FALSE;
SignalName[50]:='PRG_IO.MesIO_PTR_2_EL3024_8';	bClockIO[50]:=TRUE;	Taille[50]:=SIZEOF(PRG_IO.MesIO_PTR_2_EL3024_8);	Address[50]:=ADR(PRG_IO.MesIO_PTR_2_EL3024_8);	ReadAdsType[50]:=FALSE;	WriteAdsType[50]:=TRUE;
SignalName[51]:='PRG_IO.MesIO_PTR_2_EL1809_9';	bClockIO[51]:=TRUE;	Taille[51]:=SIZEOF(PRG_IO.MesIO_PTR_2_EL1809_9);	Address[51]:=ADR(PRG_IO.MesIO_PTR_2_EL1809_9);	ReadAdsType[51]:=FALSE;	WriteAdsType[51]:=TRUE;
SignalName[52]:='PRG_IO.MesIO_PTR_2_EL2809_10';	bClockIO[52]:=TRUE;	Taille[52]:=SIZEOF(PRG_IO.MesIO_PTR_2_EL2809_10);	Address[52]:=ADR(PRG_IO.MesIO_PTR_2_EL2809_10);	ReadAdsType[52]:=TRUE;	WriteAdsType[52]:=FALSE;
SignalName[53]:='PRG_IO.MesIO_PTR_3_EL3024_8';	bClockIO[53]:=TRUE;	Taille[53]:=SIZEOF(PRG_IO.MesIO_PTR_3_EL3024_8);	Address[53]:=ADR(PRG_IO.MesIO_PTR_3_EL3024_8);	ReadAdsType[53]:=FALSE;	WriteAdsType[53]:=TRUE;
SignalName[54]:='PRG_IO.MesIO_PTR_3_EL1809_9';	bClockIO[54]:=TRUE;	Taille[54]:=SIZEOF(PRG_IO.MesIO_PTR_3_EL1809_9);	Address[54]:=ADR(PRG_IO.MesIO_PTR_3_EL1809_9);	ReadAdsType[54]:=FALSE;	WriteAdsType[54]:=TRUE;
SignalName[55]:='PRG_IO.MesIO_PTR_3_EL2809_10';	bClockIO[55]:=TRUE;	Taille[55]:=SIZEOF(PRG_IO.MesIO_PTR_3_EL2809_10);	Address[55]:=ADR(PRG_IO.MesIO_PTR_3_EL2809_10);	ReadAdsType[55]:=TRUE;	WriteAdsType[55]:=FALSE;
SignalName[56]:='GVL_CFG.AX_PTR[1].AX_INV[1].MesDataExd';	bClockIO[56]:= TRUE;Taille[56]:=SIZEOF(GVL_CFG.AX_PTR[1].AX_INV[1].MesDataExd);	Address[56]:=ADR(GVL_CFG.AX_PTR[1].AX_INV[1].MesDataExd_IN);ReadAdsType[56]:=TRUE;	WriteAdsType[56]:=FALSE;
SignalName[57]:='GVL_CFG.AX_PTR[1].AX_INV[2].MesDataExd';	bClockIO[57]:=TRUE;	Taille[57]:=SIZEOF(GVL_CFG.AX_PTR[1].AX_INV[2].MesDataExd);	Address[57]:=ADR(GVL_CFG.AX_PTR[1].AX_INV[2].MesDataExd_IN);ReadAdsType[57]:=TRUE;	WriteAdsType[57]:=FALSE;
SignalName[58]:='GVL_CFG.AX_PTR[2].AX_INV[1].MesDataExd';	bClockIO[58]:=TRUE;	Taille[58]:=SIZEOF(GVL_CFG.AX_PTR[2].AX_INV[1].MesDataExd);	Address[58]:=ADR(GVL_CFG.AX_PTR[2].AX_INV[1].MesDataExd_IN);ReadAdsType[58]:=TRUE;	WriteAdsType[58]:=FALSE;
SignalName[59]:='GVL_CFG.AX_PTR[2].AX_INV[2].MesDataExd';	bClockIO[59]:=TRUE;	Taille[59]:=SIZEOF(GVL_CFG.AX_PTR[2].AX_INV[2].MesDataExd);	Address[59]:=ADR(GVL_CFG.AX_PTR[2].AX_INV[2].MesDataExd_IN);ReadAdsType[59]:=TRUE;	WriteAdsType[59]:=FALSE;
SignalName[60]:='GVL_CFG.AX_PTR[3].AX_INV[1].MesDataExd';	bClockIO[60]:=TRUE;	Taille[60]:=SIZEOF(GVL_CFG.AX_PTR[3].AX_INV[1].MesDataExd);	Address[60]:=ADR(GVL_CFG.AX_PTR[3].AX_INV[1].MesDataExd_IN);ReadAdsType[60]:=TRUE;	WriteAdsType[60]:=FALSE;
SignalName[61]:='GVL_CFG.AX_PTR[3].AX_INV[2].MesDataExd';	bClockIO[61]:=TRUE;	Taille[61]:=SIZEOF(GVL_CFG.AX_PTR[3].AX_INV[2].MesDataExd);	Address[61]:=ADR(GVL_CFG.AX_PTR[3].AX_INV[2].MesDataExd_IN);ReadAdsType[61]:=TRUE;	WriteAdsType[61]:=FALSE;
SignalName[62]:='GVL_CFG.AX_PTR[4].AX_INV[1].MesDataExd';	bClockIO[62]:=TRUE;	Taille[62]:=SIZEOF(GVL_CFG.AX_PTR[4].AX_INV[1].MesDataExd);	Address[62]:=ADR(GVL_CFG.AX_PTR[4].AX_INV[1].MesDataExd_IN);ReadAdsType[62]:=TRUE;	WriteAdsType[62]:=FALSE;
SignalName[63]:='GVL_CFG.AX_PTR[4].AX_INV[2].MesDataExd';	bClockIO[63]:=TRUE;	Taille[63]:=SIZEOF(GVL_CFG.AX_PTR[4].AX_INV[2].MesDataExd);	Address[63]:=ADR(GVL_CFG.AX_PTR[4].AX_INV[2].MesDataExd_IN);ReadAdsType[63]:=TRUE;	WriteAdsType[63]:=FALSE;
END_METHOD

END_PROGRAM

// ---- 00_FunctionsBlocks/AlarmManagement/FB_AlarmCodeManager.TcPOU
FUNCTION_BLOCK FB_AlarmCodeManager
////////////////// 
// Create Alarm Code from Alarms and Warnings conditions and summarize alarms
//////////////////	
VAR_INPUT
	bAlarm0				: BOOL:=FALSE; 			// Zero Alarm Condition (Optionnal only for subequipment)
	bAlarm1				: BOOL:=FALSE ; 		// First Alarm Condition  
	bAlarm2				: BOOL:=FALSE ; 		// Second Alarm Condition
	bAlarm3				: BOOL:=FALSE ; 		// Third Alarm Condition
	bAlarm4				: BOOL:=FALSE ; 		// Fourth Alarm Condition
	bAlarm5				: BOOL:=FALSE ; 		// Fifth Alarm Condition
	bAlarm6				: BOOL:=FALSE ; 		// First AlarmPermanent Condition
	bAlarm7				: BOOL:=FALSE ; 		// Second AlarmPermanent Condition
	bAlarm8				: BOOL:=FALSE ; 		// Third AlarmPermanent Condition
	bAlarm9				: BOOL:=FALSE ; 		// Fourth AlarmPermanent Condition 
	bAlarm10			: BOOL:=FALSE ; 		// Fourth AlarmPermanent Condition 
	bAlarm11			: BOOL:=FALSE ; 		// First AlarmPermanent Condition
	bAlarm12  			: BOOL:=FALSE ; 		// Second AlarmPermanent Condition
	bAlarm13			: BOOL:=FALSE ; 		// Third AlarmPermanent Condition
	bAlarm14			: BOOL:=FALSE ; 		// Fourth AlarmPermanent Condition 
	bAlarm15			: BOOL:=FALSE ; 		// Fourth AlarmPermanent Condition 

END_VAR

VAR_OUTPUT
	wAlarmCode		: WORD ; 		// 16 bit Alarm Code. 
END_VAR

VAR CONSTANT
	AlarmMask		: WORD := 2#1111111111111110 ;  // Alarm Mask 

	
END_VAR

// Reinitialize Alarm summary
wAlarmCode.0 := FALSE  ;

// Evaluate wAlarmCode
wAlarmCode.1 	:= bAlarm1 ;  
wAlarmCode.2 	:= bAlarm2 ;  
wAlarmCode.3 	:= bAlarm3 ;  
wAlarmCode.4 	:= bAlarm4 ;  
wAlarmCode.5 	:= bAlarm5 ;  
wAlarmCode.6 	:= bAlarm6 ; 
wAlarmCode.7 	:= bAlarm7 ; 
wAlarmCode.8 	:= bAlarm8 ;
wAlarmCode.9 	:= bAlarm9 ;
wAlarmCode.10 	:= bAlarm10 ; 
wAlarmCode.11 	:= bAlarm11 ; 
wAlarmCode.12 	:= bAlarm12 ; 
wAlarmCode.13 	:= bAlarm13 ; 
wAlarmCode.14 	:= bAlarm14 ; 
wAlarmCode.15 	:= bAlarm15 ; 
 
// Alarm Summarized
IF (AlarmMask AND wAlarmCode) >0 THEN
	wAlarmCode.0 := TRUE  ; 
END_IF

END_FUNCTION_BLOCK

// ---- 00_FunctionsBlocks/AlarmManagement/FB_CheckCommand.TcPOU
FUNCTION_BLOCK FB_CheckCommand
////////////////// 
// Compare command with measure and raise warning if inconsistance. 
//////////////////	
VAR_INPUT
	T					: TIME ;			// Tempo to check if command has been executed	
	bCmd				: BOOL ; 			// Input command 
	bMes				: BOOL ; 			// Measure feedback 
	bReset				: BOOL := FALSE ; 	// Reset 
	bImpulsion			: BOOL ; 			// If True , the command is done on impulsion
	
END_VAR

VAR_OUTPUT
	bWarning 			: BOOL ; 		// Warning if inconsistancy . 
	bInProgress			: BOOL ; 		// Action in Progress
	
END_VAR

VAR

	// Inconsistency detection
	R_TRIG1				: R_TRIG ; 		// Detect command
	TOF1				: TOF ; 		// Creates a falling edge T time after command detcetion	
	F_TRIG				: F_TRIG ; 		// Detect Falling edge of TOF1	
	
	F_TRIG2				: F_TRIG ; 		// Detect falling edge of feedback measure
	TOF2				: TOF ; 		// Creates  a falling edge T time after Feedback measure ended detcetion
 
	TON					: TON ; 		// Tempo in case of bistable functuion

	// Reset management 	
	TOF_Reset			: TOF;			// Hold Reset command afetr reset to inhibate future warnings
	RS_Reset			: RS;			// Maintain reset command
	
END_VAR

IF bReset THEN
	bWarning 	:= FALSE ; 
END_IF

// Reset management 
TOF_Reset(IN:= bReset ,PT :=T);
RS_Reset(SET := bCmd,RESET1 := bReset) ; 


IF bImpulsion THEN 
	// Command is an impulsion
	R_TRIG1(CLK := bCmd) ; 
	TOF1(IN:=R_TRIG1.Q , PT:=T) ;
	F_TRIG(CLK:=TOF1.Q);		

	F_TRIG2(CLK := bMes) ;  
	TOF2(IN:=F_TRIG2.Q , PT:=T) ; 

ELSE
	// Command is a bistable function
	TON(IN:=bCmd , PT:= T);
END_IF

// Reset to False "InProgress" if Reset command or if command has been executed . 
bInProgress :=  ((TON.ET < TON.PT) AND (TON.ET>T#0S) OR (TOF1.ET < TOF1.PT) AND (TOF1.ET>T#0S)) AND NOT bMes AND RS_Reset.Q1  ; 

// Inconsistency detection
IF ((F_TRIG.Q AND NOT TOF2.Q AND NOT bMes) OR (TON.Q AND NOT bMes)) AND NOT TOF_Reset.Q  THEN
	bWarning := TRUE ; 
END_IF

END_FUNCTION_BLOCK

// ---- 00_FunctionsBlocks/AlarmManagement/FB_CheckSetpt.TcPOU
FUNCTION_BLOCK FB_CheckSetpt
////////////////// 
// Compare SetPoint with measure and raise warning if inconsistance.
// The measure has to be within a range around the setpoint after a certain delay  . 
//////////////////	
VAR_INPUT
	T					: TIME ;		// Time to reacbh the range . 
	Tolerance			: INT := 5 ; 	// (%) Tolerance Window  
	Range 				: REAL ; 		// Maximal Range of the Setpoint
	bTrigger			: BOOL ; 		// Moment from which the setpoint is taken as reference
	bSetpt				: REAL ; 		// Input setpoint 
	bMes				: REAL ; 		// Measure feedback 
	bReset				: BOOL ; 		// Reset 
	
END_VAR

VAR_OUTPUT
	bWarning 			: BOOL ; 		// Warning if inconsistancy . 
	
END_VAR
VAR
	R_TRIG				: R_TRIG ; 		// Detect Trigger activation
	TOF					: TOF ; 		// Creates a falling edge T time after trigger activation
	F_TRIG				: F_TRIG ; 		// Detect end of timer. 
	
END_VAR

// Inconsistency detection

R_TRIG(CLK := bTrigger)  ;
TOF(IN := R_TRIG.Q , PT := T); 
F_TRIG(CLK := TOF.Q) ;


IF F_TRIG.Q AND ABS(bMes-bSetpt)>Tolerance/100*Range  THEN
	bWarning := TRUE ; 
END_IF

// Reset warning
IF bReset THEN
	bWarning := FALSE ; 
END_IF

END_FUNCTION_BLOCK

// ---- 00_FunctionsBlocks/AlarmManagement/FB_DetectFixedValue.TcPOU
FUNCTION_BLOCK FB_DetectFixedValue
VAR_INPUT
	IN_Addr			: POINTER TO BYTE;			// Adr of the variable to  analyse
	IN_EmptyStruct	: POINTER TO BYTE;			// Adr of a null variable on which I input the compared value
	IN_Size			: UINT;						// Size of the variable to analyse
	IN_Duration		: TIME;						// Duration after which an alarm is raised
END_VAR
VAR_OUTPUT
	OUT_bStatic		: BOOL;						// Value has been static for more than IN_Duration time
END_VAR
VAR
	TON_CMP			: TON;
	bFixed			: BOOL;
END_VAR

bFixed :=  MEMCMP(pBuf1 := IN_Addr, pBuf2 := IN_EmptyStruct, n := IN_SIZE)=0;

TON_CMP(IN := bFixed, PT := IN_Duration, Q => OUT_bStatic);

IF NOT bFixed THEN
	MEMCPY(destAddr := IN_EmptyStruct, srcAddr := IN_Addr, n := IN_Size);
END_IF

END_FUNCTION_BLOCK

// ---- 00_FunctionsBlocks/AlarmManagement/FB_DetectFlicker.TcPOU
FUNCTION_BLOCK FB_DetectFlicker
// Detect if a booleean variable is flickering 

VAR_INPUT
	IN_VAR			: BOOL;						// Boolean input to analyze
	IN_Window		: TIME := T#5S;				// Time Window during which I check the number of value change
	IN_Count		: UINT;						// Maximum number of change for the tiume duration 

END_VAR
VAR_OUTPUT
	OUT_bFlicker		: BOOL;					// Value is considered as flickering
END_VAR
VAR
	COUNT 			: CTU ; 
	TON				: TON ; 
END_VAR

TON(IN:= TRUE , PT:= IN_Window ) ; 

IF COUNT.CV > IN_Count THEN 
	OUT_bFlicker := TRUE ; 
ELSIF COUNT.CV < IN_Count AND TON.Q THEN  
	OUT_bFlicker := FALSE ; 
END_IF	
	
COUNT(CU:= IN_VAR , PV:= 1000 , RESET:=TON.Q)  ; 

IF TON.Q THEN 
	TON(IN:= FALSE ) ; 
END_IF

END_FUNCTION_BLOCK

// ---- 00_FunctionsBlocks/AlarmManagement/FB_HeartBeatMasterBackup.TcPOU
FUNCTION_BLOCK FB_HeartBeatMasterBackup
//////////////////
// heart beat detector using ADS . 
//////////////////

VAR_INPUT PERSISTENT
	// Parameters of the Object (instance specific) 
	ParamTempoImpulsion3		: TIME := T#500MS ;			// (s) Config : Tempo command impulsion
	ParamTimeout				: TIME  := T#100MS ;				// (Time) Timeout for modbus reading
	                                                    
END_VAR                                                 
                                                        
VAR_INPUT                                               
	//M_Backup Variables//       
//{attribute 'OPC.UA.DA' := '1'}                       
	sNetId 				   		: STRING(20);      					// (NA) ADS device identification Adress
	nPort				  		: UINT := 851;					    // (NA) ADS device Port
	IdxGroup					: UDINT:=16#4020;		// Counter TMC Group Index
	IdxOff						: UDINT:=4; 		// Counter TMC Offset Index
END_VAR                                                             
                                                                    
VAR_OUTPUT                                                          
	bHeartBeat					: BOOL := FALSE;					// (NA) Heart beat detector : False if complete loss of communication with the master
	nCounter                     AT%Q* : BYTE;					    // (NA) Variable to increment in the master	
END_VAR                                                 
                                                        
VAR                                                     
	//M_Backup Variables//                              
	ADSREADEX1                  : ADSREADEX;						// (NA) Functionnal Block to request data from an ADS device
	                                                    			
	TP1							: TP ; 							// (NA) Tempo to define ADS Reading Frequency 
	R_TRIG1						: R_TRIG;							// (NA) Tempo Rising edge detection for ADS Reading
	TON_Freeze					: TON;                                                    			
	ClockRead					: BOOL;								// (NA) ADS reading Clock
	nResult  					: BYTE;            					// (NA) Variable in which the read data have to be stored
	nResult_Temp				: BYTE;	
	bBusy						: BOOL;                             // (NA) Busy Flag
	bError						: BOOL;            					// (NA) Error Flag
	ErrorId						: UDINT;           					// (NA) Error Id returned by FB (see ADS error Code)
	//M_Master Variables//  

	CountError					: UINT ;
	CountOK						: UINT ; 
	
END_VAR

METHOD M_Backup

VAR
	// Method local variables (reinitialized at each cycle) 

END_VAR
TP1(IN:= NOT TP1.Q,PT:=ParamTempoImpulsion3);
R_TRIG1(CLK:=TP1.Q,Q=>ClockRead);

ADSREADEX1(NETID:=sNetId,
		   PORT:=nPort,
		   IDXGRP:=IdxGroup,
		   IDXOFFS:=IdxOff,
		   LEN:=1,
		   READ:=ClockRead,
		   DESTADDR:=ADR(nResult),
		   TMOUT:=ParamTimeout,
		   BUSY=>bBusy,
		   ERR=>bError,
		   ERRID=>ErrorId);
		   

TON_Freeze(IN:= (nResult =nResult_Temp), PT:=ParamTempoImpulsion3 ) ; 		    	   

// Case : after a restart of the master , the Counter  = 0 fixed . Then the slave detects a change 
		   
IF NOT bBusy AND bError THEN
	// IF ADS fails ( Beckhoff is down, not answering ADS) 
	CountError := CountError +1 ; 

ELSIF NOT bBusy AND NOT bError AND NOT TON_Freeze.Q  THEN
	// Return to PLC master OK . OR  Data is incrementing
	CountOK := CountOK+1 ; 
	//bHeartBeat:=TRUE;
	CountError := 0 ; 
	nResult_Temp := nResult ;
ELSIF NOT bBusy AND NOT bError AND TON_Freeze.Q THEN 
	// Counter is frozen ( Master untime stopped , or no stable operation ) 
	bHeartBeat:=FALSE;
	CountError := 0 ; 
	CountOK:= 0 ; 
	nResult_Temp := nResult ;
END_IF


IF CountError > 2  THEN 
	bHeartBeat:=FALSE;
	CountOK:= 0 ; 
ELSIF CountOK>=2 THEN 
	// Return to PLC MAster OK ( makes sure that the change of variables is steady ) 
	bHeartBeat:=TRUE;
END_IF
END_METHOD

METHOD M_Master

VAR
	// Method local variables (reinitialized at each cycle) 
END_VAR
IF MAIN.CalStableOp_G THEN 
	nCounter:=MAX(1,nCounter +1); 			// Return to Master PLC possible . Safe operation
	
ELSE
	
	nCounter:=0;
	
END_IF
END_METHOD

END_FUNCTION_BLOCK

// ---- 00_FunctionsBlocks/AlarmManagement/FB_UnknownEvent.TcPOU
FUNCTION_BLOCK FB_UnknownEvent
////////////////// 
// Detect an event that is not the result of an internal command, or an external event
//////////////////	
VAR_INPUT
	IN_TempoAfterCommand					: TIME ;					// Tempo between internal command and event
	IN_TempoReadExternalEvent					: TIME ;					// Tempo to read the external event
	
	IN_InternalCommand				: BOOL ; 			// Internal command that normally trigers the event 
	IN_ExternalEvent				: BOOL ; 			// External Event that normally explains the Event (to be read after the event)
	
	IN_Event						: BOOL ; // Event that occur
	
	bReset				: BOOL := FALSE ; 	// Reset 
	
END_VAR

VAR_OUTPUT
	OUT_Unknown 			: BOOL ; 		// Flag to TRUE is the event is unknown ( neither related to the command, or an external event that is known) 
	
END_VAR

VAR
	FB_CheckCommand : FB_CheckCommand ;
	// Inconsistency detection
	R_TRIG1				: R_TRIG ; 		// Detect command
	TOF1				: TOF ; 		// Creates a falling edge T time after command detcetion	
	F_TRIG				: F_TRIG ; 		// Detect Falling edge of TOF1	
	
	F_TRIG2				: F_TRIG ; 		// Detect falling edge of feedback measure
	TOF2				: TOF ; 		// Creates  a falling edge T time after Feedback measure ended detcetion
 
	TON					: TON ; 		// Tempo in case of bistable functuion

	// Reset management 	
	TOF_Reset			: TOF;			// Hold Reset command afetr reset to inhibate future warnings
	RS_Reset			: RS;			// Maintain reset command
	
	R_TRIG2: R_TRIG;
	CalNotLinkedToCommand: BOOL;
END_VAR


R_TRIG1(CLK := IN_InternalCommand) ; 

TOF1(IN:=R_TRIG1.Q , PT:=IN_TempoAfterCommand) ;
F_TRIG(CLK:=TOF1.Q);		

R_TRIG2(CLK := IN_Event) ; 


CalNotLinkedToCommand :=  NOT TOF1.Q AND R_TRIG2.Q ;
 
FB_CheckCommand(T:= IN_TempoReadExternalEvent , bCmd := CalNotLinkedToCommand , bMes := IN_ExternalEvent , bReset := bReset , bImpulsion := TRUE ) ; 
OUT_Unknown := FB_CheckCommAND.bWarning  ;

END_FUNCTION_BLOCK

// ---- 00_FunctionsBlocks/AlarmManagement/FUN_Alarms_CSV.TcPOU
PROGRAM FUN_Alarms_CSV
////////////////// 
// Save Alarms in a CSV File locally. 
//////////////////	
VAR_INPUT
	ParamSeparateur			: STRING := ';';				// Separator for the CSV file
	ParamExtension			: STRING(255) := '.csv';				// File extension
	FIFO					: FB_DBDatasetFifo;	// Buffer that contains all the alarms to be written in the file. 
	
END_VAR
VAR_OUTPUT
	
END_VAR
VAR
	format_string				: FB_Formatstring;
	CalDate						: T_MaxString;
	
	// Alarm management 
		bWriteAlarm				: BOOL;				// Writing CSV File failed 
		TON_WritealarmFile		: TON;				// Tempo to detect error in file creation.  
		
		
	// Data processing 
	MesData				: ServerCSV ;			//  Server info
	CalFileName			: STRING;				// Name of csv file 
	
	//Time Values 
	
	//Test existence file 
	FindFile 			: FB_EnumFindFileEntry ;
	FileInfo			: ST_FindFileEntry;
	bFileOK				: BOOL:= TRUE ;

	//Initial File creation 
	GetHostName			: FB_GetHostName;
	WriteFile			: FB_WriteFile;
	bStartWrite			: BOOL;
	bInitWrite			: BOOL;
	
	//Initial File creation 
	InitLine			: T_MaxString;
	LastInitLine		: T_MaxString;
	WelcomeMessage 		: T_MaxString := 'Daily alarms file';
	ForDay				: T_MaxString := 'for day :';
	ForPlant	 		: T_MaxString := 'for plant : ';
	NewLineVar			: T_MaxString := '$L $00';
	TimeStampVar		: T_MaxString := 'TimeStamp;AlarmsID;Description;Activated;Acknowledged;Level;$L$00';
	MessageInitial		: ARRAY[1..10] OF STRING(255);
	MessageInitial_Null	: ARRAY[1..10] OF STRING(255);
	bInitWriting		: BOOL;
	len_to_write		: INT;
	len_to_add			: INT;

	// Write File
	LineToWrite			: STRING(1000);

	// General variables
		bInit 			: BOOL;
		MesTimeStamp 	: STRING(19);				// Timestamp of the alarm
		bOutCompleted 	: RS;						// Writing file is completed
	
	//TABLEAU
		CalTimeStamp: STRING(255);				// Timestamp formatted

END_VAR

IF NOT bInit THEN
	M_Init();
END_IF

M_AlarmManager();

format_string(
	sFormat := 'ALARMS_%0.2d-%0.2d-%0.2d%s', 
	arg1 := F_WORD(in:=CalLocalTimeStruct.wYear),	arg2 := F_WORD(in:=CalLocalTimeStruct.wMonth),	arg3 := F_WORD(in:=CalLocalTimeStruct.wDay),
	arg4 := F_STRING(in:=ParamExtension),
	sOut => CalFileName
);

format_string(
	sFormat := '%0.2d-%0.2d-%0.2d', 
	arg1 := F_WORD(in:=CalLocalTimeStruct.wYear),	arg2 := F_WORD(in:=CalLocalTimeStruct.wMonth),	arg3 := F_WORD(in:=CalLocalTimeStruct.wDay),
	sOut => CalDate
);

InitLine := concat(str1:=WelcomeMessage, STR2:= concat(str1:=
	ParamSeparateur, str2:=concat(STR1:=ForDay, STR2:=concat(str1:= ParamSeparateur, STR2:= concat(str1:= 
	CalDate,str2:=concat(str1:= ParamSeparateur, str2 := CONCAT(str1:=
	ForPlant,str2:=Concat(str1:=ParamSeparateur, str2:= CONCAT(str1:= GetHostName.sHostName, str2:=ParamSeparateur)
))))))));

IF InitLine <> LastInitLine OR InitLine = '' THEN
	LastInitLine := InitLine;
	bInitWriting := TRUE;
END_IF
		
//Test Existence File
IF FUN_CreateDir_CSV.bDirOk THEN
	FindFile
	(
		sNetId := '',
		sPathName := concat(FUN_CreateDir_CSV.AX_DirNames[2],CalFileName),
		eCmd := eEnumCmd_First,
		bExecute := TRUE,
		tTimeout := T#3S,
		stFindFile => FileInfo
	);
	
MesData.TimeCreation 	:= FILETIME_TO_SYSTEMTIME(filetime := FileInfo.creationTime);
MesData.TimeModif	 	:= FILETIME_TO_SYSTEMTIME(filetime := FileInfo.lastWriteTime);
	
MesData.FileSize  		:= ULARGE_TO_ULINT(in := FileInfo.fileSize);
	IF NOT FindFile.bBusy THEN
		FindFile(bExecute := FALSE);
		bFileOK := MesData.FileSize > 0 ; 
	END_IF
	
	
	IF NOT FindFile.bBusy AND NOT bFileOK AND bInitWriting THEN
	// Write File Initial
		bInitWriting := TRUE;
		// je réinitialise les longueurs
		len_to_write := 0;
		MessageInitial := MessageInitial_Null;
		MEMCPY(destAddr := ADR(MessageInitial)+len_to_write, srcAddr := ADR(InitLine), n := len(InitLine));
		len_to_add := len(InitLine);			len_to_write := len_to_write + len_to_add;
		
		MEMCPY(destAddr := ADR(MessageInitial)+len_to_write, srcAddr := ADR(NewLineVar), n := len(NewLineVar));
		len_to_add := len(NewLineVar);			len_to_write := len_to_write + len_to_add;
		
		MEMCPY(destAddr := ADR(MessageInitial)+len_to_write, srcAddr := ADR(TimeStampVar), n := len(TimeStampVar));
		len_to_add := len(TimeStampVar);		len_to_write := len_to_write + len_to_add;
		
		WriteFile
		(
			InStart := TRUE,
			InDirFile := concat(FUN_CreateDir_CSV.AX_DirNames[2], CalFileName),
			InAmsId := '', 
			InPMessage := ADR(MessageInitial),
			InLMessage := len_to_write
		);
		
		IF WriteFile.OutCompleted THEN
			WriteFile(InStart := FALSE);
			bInitWriting := FALSE;
		END_IF
	END_IF
	
	
	IF bFileOK AND MesData.FileSize < 100000000 AND fifo.nCount > 0 AND NOT bInitWriting THEN
		fifo.A_Get();	// Unpile the buffer to get the next alarm to write. 
		
		MesTimeStamp := CONCAT(REPLACE(STR1:= left(str := FIFO.Out.TimeStamp_Act, 19), STR2 := ' ', L := 1, P := 11), ' ') ;	// Get Timestamp of the activation or desactivation of the alarm
		ReplaceAll( In_StringTosearch := MesTimeStamp, In_StringToFind := '/', IN_StringToReplace := '-', OUT_StringToSearch => CalTimeStamp);
		
		// Create line content
		LineToWrite := Concat(CalTimeStamp, ParamSeparateur);
		LineToWrite := concat(LineToWrite, Concat(STR1 := UINT_TO_STRING(FIFO.Out.ID) ,ParamSeparateur));
		LineToWrite := concat(LineToWrite, Concat(STR1 := FIFO.Out.Message ,ParamSeparateur));
		LineToWrite := Concat(STR1 := LineToWrite, STR2 := Concat(STR1 := BOOL_TO_STRING( FIFO.Out.Value), STR2 := ParamSeparateur));
		LineToWrite:= Concat(STR1 := LineToWrite, Concat(STR1 := BOOL_TO_STRING( FIFO.Out.Ack), STR2 := ParamSeparateur)); 
		LineToWrite:= Concat(STR1 := LineToWrite, Concat(STR1 := UINT_TO_STRING( FIFO.Out.Alarms_LVL), STR2 := ParamSeparateur)); 
		LineToWrite := Concat(LineToWrite, '$L$00');
		
		// Write File
		WriteFile
		(
			InStart := TRUE,
			InDirFile := concat(FUN_CreateDir_CSV.AX_DirNames[2], CalFileName),
			InAmsId := '', 
			InPMessage := ADR(LineToWrite),
			InLMessage := LEN(LineToWrite)
		);
		IF NOT WriteFile.OutBusy AND NOT WriteFile.OutError AND WriteFile.OutCompleted THEN
			// File has been writen successfully
			fifo.A_Remove();
			WriteFile(InStart := FALSE);
			bWriteAlarm	:= FALSE ;
		ELSIF WriteFile.OutError THEN 
			// In case of writing error, try again to write the alarm. 
			bWriteAlarm	:= TRUE ;
			WriteFile(InStart := FALSE);
		END_IF
	END_IF
END_IF

METHOD M_AlarmManager
VAR

	FB_AlarmCodeManager			: FB_AlarmCodeManager ;

END_VAR

TON_WritealarmFile(IN:= NOT bFileOK  , PT:= T#10S  ) ;


// ALARM CODE //
	FB_AlarmCodeManager(
		bAlarm1			:= bWriteAlarm	  ,				// Write CSV Alarm
		bAlarm2			:= fifo.bOverwrite   ,			// Overflow buffer
		bAlarm3			:= TON_WritealarmFile.Q   ,		// Can not create CSV Alarm file 
		bAlarm4			:= FALSE	 ,					//
		bAlarm5			:= FALSE	,					// 
		bAlarm6			:= FALSE,									//
		bAlarm7			:= FALSE,                                   //
		bAlarm8			:= FALSE,                                   //
		bAlarm9			:= FALSE,                                   //
		bAlarm10		:= FALSE,                                   //
		bAlarm11		:= FALSE,									//
		bAlarm12		:= FALSE,                                   //
		bAlarm13		:= FALSE,                                   //
		bAlarm14		:= FALSE,                                   //
		bAlarm15		:= FALSE,                                   //
		wAlarmCode		=>MesData.MesAlarmCode);
END_METHOD

METHOD M_Init

VAR
	LL	: SINT;
	KK 	: SINT;
	InStruct : ST_ValuesAlarms;
END_VAR
// Create a first alarm after new code activation or PLC restart
//	FIFO.A_Get();
//	FIFO.A_Remove();
	bInit := TRUE;


	GetHostName(bExecute := FALSE);
	GetHostName(bExecute := TRUE);
END_METHOD

END_PROGRAM

// ---- 00_FunctionsBlocks/Fifo/FB_DBDatasetFifo.TcPOU
FUNCTION_BLOCK FB_DBDatasetFifo
VAR_INPUT
    bOverwrite : BOOL;
    In         : ST_ValuesAlarms;
END_VAR
VAR_OUTPUT
    bOk        : BOOL;
    nCount     : UDINT;
    nLoad      : UDINT;
    Out        : ST_ValuesAlarms;
END_VAR
VAR
    arrBuffer  : ARRAY[0..Max_buffer_size_G] OF BYTE; (* Buffer memory used by FB_MemRingBuffer function block *)
    fbBuffer   : FB_MemRingBuffer;
END_VAR

ACTION A_Add:
fbBuffer.A_AddTail(pWrite := ADR(in),
						   cbWrite:=SIZEOF(in),
						   pBuffer:=ADR(arrBuffer),
						   cbBuffer:=SIZEOF(arrBuffer),
						   bOK=>bOK,
						   nCount =>nCount);
IF NOT bOK THEN 
	IF bOverwrite THEN
		fbBuffer.A_RemoveHead();(*remove one oldest entry*)
		fbBuffer.A_AddTail(bOK => bOk,nCount => nCount);
	END_IF
END_IF

nload := (fbbuffer.cbSize * 100)/(Max_buffer_size_G);
END_ACTION

ACTION A_Get:
fbBuffer.A_GetHead(pWrite := ADR(out),
						   cbWrite:=SIZEOF(out),
						   pBuffer:=ADR(arrBuffer),
						   cbBuffer:=SIZEOF(arrBuffer),
						   bOK=>bOK,
						   nCount =>nCount);
nload := (fbbuffer.cbSize * 100)/(Max_buffer_size_G);
END_ACTION

ACTION A_Remove:
fbBuffer.A_RemoveHead(pRead:=ADR(out),
						cbRead:=SIZEOF(out),
						pBuffer:=ADR(arrBuffer),
						cbBuffer:=SIZEOF(arrBuffer),
						bOK=>bOK,
						nCount =>nCount);
nload := (fbbuffer.cbSize * 100)/(Max_buffer_size_G);
END_ACTION

ACTION A_Reset:
MEMSET(ADR(arrBuffer),0,SIZEOF(arrBuffer)); (*reset internal buffer*)
fbBuffer.A_Reset(bOK=>bOK,nCount=>ncount);
nload := (fbbuffer.cbSize * 100)/(Max_buffer_size_G);
END_ACTION

END_FUNCTION_BLOCK

// ---- 00_FunctionsBlocks/DataProcessing/WriteFile/FB_WriteFile.TcPOU
FUNCTION_BLOCK FB_WriteFile

VAR_INPUT 
	InDirFile : STRING(1000);
	InAmsId : T_AmsNetID :='';
	InPMessage: POINTER TO BYTE;
	InLMessage: UDINT;
	InStart : BOOL;
	InMode : DWORD := 16#4;	// Append Mode . 
END_VAR

VAR_OUTPUT
	OutBusy 	: BOOL;
	OutError 	: BOOL;
	OutErrorId 	: STRING;
	cbWritten 	: UDINT;
	OutCompleted : BOOL;
END_VAR

VAR 
MesDataExd: LoggerCSV;
	FileHandle 	: UINT;
	select		: INT;
	AX_ErrorId	: ARRAY[1..NbSteps] OF UDINT;
	AX_Error 	: ARRAY[1..NbSteps] OF BOOL;
	OpenFile 	: FB_FileOpen;
	CloseFile 	: FB_FileClose;
	WriteFile 	: FB_FileWrite;
	TextToWrite : STRING(255);
	nSeekPos 	: DINT;
	i 			: UINT;
	bCompleted	: BOOL;
	Trigger		: R_TRIG;
END_VAR

VAR CONSTANT
	NbSteps 	: UINT := 3;
END_VAR

OutCompleted := FALSE;
CASE select OF
	0: // Initialize
		Trigger(CLK := InStart);
		IF Trigger.Q THEN
			select := 1;
			OutBusy := TRUE;
			OutError := FALSE;
			OutErrorId :='';
		END_IF
	1:
		OpenFile(sNetId := InAmsId, 
			sPathName := InDirFile,
			nMode := InMode,
			ePath := Path_generic,
			bExecute := TRUE,
			hFile => FileHandle,
			nErrId => AX_ErrorId[Select],
			bError => AX_Error[Select]
		);
		IF NOT(OpenFile.bBusy) THEN
 			IF NOT(OpenFile.bError) THEN
				select := select+1;
				OpenFile(bExecute := FALSE);
			ELSE
				select := -1;
			END_IF
		END_IF

